LIN {X 0,Y 119.724,Z 602.099,A -85,B 0,C 180,E1 -25798.109,E2 -25798.109} C_VEL
LIN {X 0,Y 115.833,Z 604.315,A -85,B 0,C 180,E1 -25804.868,E2 -25804.868} C_VEL
LIN {X 0,Y 114.441,Z 604.822,A -85,B 0,C 180,E1 -25808.379,E2 -25808.379} C_VEL
LIN {X 0,Y 113.363,Z 604.891,A -85,B 0,C 180,E1 -25811.943,E2 -25811.943} C_VEL
LIN {X 0,Y 112.315,Z 603.854,A -85,B 0,C 180,E1 -25819.18,E2 -25819.18} C_VEL
LIN {X 0,Y 112.318,Z 602.743,A -85,B 0,C 180,E1 -25822.811,E2 -25822.811} C_VEL
LIN {X 0,Y 112.71,Z 601.178,A -85,B 0,C 180,E1 -25826.425,E2 -25826.425} C_VEL
LIN {X 0,Y 113.504,Z 598.082,A -85,B 0,C 180,E1 -25831.774,E2 -25831.774} C_VEL
LIN {X 0,Y 115.031,Z 593.941,A -85,B 0,C 180,E1 -25837.019,E2 -25837.019} C_VEL
LIN {X 0,Y 117.787,Z 587.628,A -85,B 0,C 180,E1 -25842.929,E2 -25842.929} C_VEL
LIN {X 0,Y 120.92,Z 580.766,A -85,B 0,C 180,E1 -25847.766,E2 -25847.766} C_VEL
LIN {X 0,Y 124.856,Z 572.161,A -85,B 0,C 180,E1 -25852.33,E2 -25852.33} C_VEL
LIN {X 0,Y 128.63,Z 563.345,A -85,B 0,C 180,E1 -25855.918,E2 -25855.918} C_VEL
LIN {X 0,Y 132.921,Z 552.472,A -85,B 0,C 180,E1 -25859.279,E2 -25859.279} C_VEL
LIN {X 0,Y 136.5,Z 541.503,A -85,B 0,C 180,E1 -25861.852,E2 -25861.852} C_VEL
LIN {X 0,Y 139.764,Z 529.243,A -85,B 0,C 180,E1 -25864.015,E2 -25864.015} C_VEL
LIN {X 0,Y 142.165,Z 517.629,A -85,B 0,C 180,E1 -25865.511,E2 -25865.511} C_VEL
LIN {X 0,Y 143.999,Z 504.981,A -85,B 0,C 180,E1 -25866.631,E2 -25866.631} C_VEL
LIN {X 0,Y 145.261,Z 489.73,A -85,B 0,C 180,E1 -25867.417,E2 -25867.417} C_VEL
LIN {X 0,Y 147.355,Z 457.951,A -85,B 0,C 180,E1 -25868.753,E2 -25868.753} C_VEL
LIN {X 0,Y 142.937,Z 448.506,A -85,B 0,C 180,E1 -25871.155,E2 -25871.155} C_VEL
LIN {X 0,Y 138.396,Z 440.269,A -85,B 0,C 180,E1 -25873.793,E2 -25873.793} C_VEL
LIN {X 0,Y 132.869,Z 431.292,A -85,B 0,C 180,E1 -25877.377,E2 -25877.377} C_VEL
LIN {X 0,Y 128.994,Z 425.855,A -85,B 0,C 180,E1 -25880.194,E2 -25880.194} C_VEL
LIN {X 0,Y 126.809,Z 422.709,A -85,B 0,C 180,E1 -25881.964,E2 -25881.964} C_VEL
LIN {X 0,Y 124.311,Z 419.474,A -85,B 0,C 180,E1 -25884.142,E2 -25884.142} C_VEL
LIN {X 0,Y 123.333,Z 418.034,A -85,B 0,C 180,E1 -25885.079,E2 -25885.079} C_VEL
LIN {X 0,Y 120.711,Z 415.377,A -85,B 0,C 180,E1 -25887.661,E2 -25887.661} C_VEL
LIN {X 0,Y 119.493,Z 412.941,A -85,B 0,C 180,E1 -25889.14,E2 -25889.14} C_VEL
LIN {X 0,Y 116.855,Z 411.214,A -85,B 0,C 180,E1 -25892.217,E2 -25892.217} C_VEL
LIN {X 0,Y 115.382,Z 409.029,A -85,B 0,C 180,E1 -25894.399,E2 -25894.399} C_VEL
LIN {X 0,Y 114.918,Z 407.137,A -85,B 0,C 180,E1 -25895.48,E2 -25895.48} C_VEL
LIN {X 0,Y 114.999,Z 407.157,A -85,B 0,C 180,E1 -25898.488,E2 -25898.488} C_VEL
LIN {X 0,Y 115.147,Z 407.106,A -85,B 0,C 180,E1 -25905.868,E2 -25905.868} C_VEL
LIN {X 0,Y 115.383,Z 407.111,A -85,B 0,C 180,E1 -25909.47,E2 -25909.47} C_VEL
LIN {X 0,Y 115.525,Z 407.056,A -85,B 0,C 180,E1 -25916.511,E2 -25916.511} C_VEL
LIN {X 0,Y 115.992,Z 407.035,A -85,B 0,C 180,E1 -25919.999,E2 -25919.999} C_VEL
LIN {X 0,Y 115.386,Z 407.107,A -85,B 0,C 180,E1 -25926.996,E2 -25926.996} C_VEL
LIN {X 0,Y 115.282,Z 407.118,A -85,B 0,C 180,E1 -25932.737,E2 -25932.737} C_VEL
LIN {X 0,Y 115.102,Z 407.186,A -85,B 0,C 180,E1 -25935.266,E2 -25935.266} C_VEL
LIN {X 0,Y 115.765,Z 409.428,A -85,B 0,C 180,E1 -25936.533,E2 -25936.533} C_VEL
LIN {X 0,Y 117.512,Z 411.742,A -85,B 0,C 180,E1 -25938.977,E2 -25938.977} C_VEL
LIN {X 0,Y 119.662,Z 413.079,A -85,B 0,C 180,E1 -25941.406,E2 -25941.406} C_VEL
LIN {X 0,Y 121.217,Z 416.052,A -85,B 0,C 180,E1 -25943.241,E2 -25943.241} C_VEL
LIN {X 0,Y 123.842,Z 418.627,A -85,B 0,C 180,E1 -25945.752,E2 -25945.752} C_VEL
LIN {X 0,Y 126.211,Z 422.141,A -85,B 0,C 180,E1 -25947.91,E2 -25947.91} C_VEL
LIN {X 0,Y 127.644,Z 423.794,A -85,B 0,C 180,E1 -25949.072,E2 -25949.072} C_VEL
LIN {X 0,Y 133.069,Z 431.531,A -85,B 0,C 180,E1 -25953.113,E2 -25953.113} C_VEL
LIN {X 0,Y 135.417,Z 435.627,A -85,B 0,C 180,E1 -25954.72,E2 -25954.72} C_VEL
LIN {X 0,Y 139.89,Z 445.297,A -85,B 0,C 180,E1 -25957.641,E2 -25957.641} C_VEL
LIN {X 0,Y 143.764,Z 455.4,A -85,B 0,C 180,E1 -25960.032,E2 -25960.032} C_VEL
LIN {X 0,Y 145.961,Z 461.997,A -85,B 0,C 180,E1 -25961.35,E2 -25961.35} C_VEL
LIN {X 0,Y 146.48,Z 475.088,A -85,B 0,C 180,E1 -25962.418,E2 -25962.418} C_VEL
LIN {X 0,Y 143.833,Z 511.707,A -85,B 0,C 180,E1 -25963.987,E2 -25963.987} C_VEL
LIN {X 0,Y 141.833,Z 525.299,A -85,B 0,C 180,E1 -25965.008,E2 -25965.008} C_VEL
LIN {X 0,Y 139.153,Z 538.159,A -85,B 0,C 180,E1 -25966.518,E2 -25966.518} C_VEL
LIN {X 0,Y 135.501,Z 550.822,A -85,B 0,C 180,E1 -25968.602,E2 -25968.602} C_VEL
LIN {X 0,Y 131.606,Z 562.106,A -85,B 0,C 180,E1 -25971.137,E2 -25971.137} C_VEL
LIN {X 0,Y 128.058,Z 571.239,A -85,B 0,C 180,E1 -25973.846,E2 -25973.846} C_VEL
LIN {X 0,Y 124.131,Z 580.605,A -85,B 0,C 180,E1 -25977.462,E2 -25977.462} C_VEL
LIN {X 0,Y 120.672,Z 588.035,A -85,B 0,C 180,E1 -25981.103,E2 -25981.103} C_VEL
LIN {X 0,Y 119.023,Z 592.301,A -85,B 0,C 180,E1 -25983.714,E2 -25983.714} C_VEL
LIN {X 0,Y 116.084,Z 599.069,A -85,B 0,C 180,E1 -25988.7,E2 -25988.7} C_VEL
LIN {X 0,Y 113.919,Z 604.457,A -85,B 0,C 180,E1 -25993.882,E2 -25993.882} C_VEL
LIN {X 0,Y 112.781,Z 608.657,A -85,B 0,C 180,E1 -25999.226,E2 -25999.226} C_VEL
LIN {X 0,Y 112.429,Z 610.864,A -85,B 0,C 180,E1 -26002.818,E2 -26002.818} C_VEL
LIN {X 0,Y 112.472,Z 613.501,A -85,B 0,C 180,E1 -26008.801,E2 -26008.801} C_VEL
LIN {X 0,Y 112.48,Z 614.275,A -85,B 0,C 180,E1 -26011.386,E2 -26011.386} C_VEL
LIN {X 0,Y 112.406,Z 615.185,A -85,B 0,C 180,E1 -26017.183,E2 -26017.183} C_VEL
LIN {X 0,Y 113.533,Z 614.858,A -85,B 0,C 180,E1 -26024.336,E2 -26024.336} C_VEL
LIN {X 0,Y 116.286,Z 613.013,A -85,B 0,C 180,E1 -26031.261,E2 -26031.261} C_VEL
LIN {X 0,Y 118.378,Z 611.46,A -85,B 0,C 180,E1 -26034.556,E2 -26034.556} C_VEL
LIN {X 0,Y 122.171,Z 608.364,A -85,B 0,C 180,E1 -26039.272,E2 -26039.272} C_VEL
LIN {X 0,Y 126.647,Z 604.233,A -85,B 0,C 180,E1 -26043.705,E2 -26043.705} C_VEL
LIN {X 0,Y 132.788,Z 597.948,A -85,B 0,C 180,E1 -26048.453,E2 -26048.453} C_VEL
LIN {X 0,Y 138.847,Z 591.139,A -85,B 0,C 180,E1 -26052.118,E2 -26052.118} C_VEL
LIN {X 0,Y 145.543,Z 582.699,A -85,B 0,C 180,E1 -26055.417,E2 -26055.417} C_VEL
LIN {X 0,Y 149.922,Z 576.362,A -85,B 0,C 180,E1 -26057.334,E2 -26057.334} C_VEL
LIN {X 0,Y 152.189,Z 572.121,A -85,B 0,C 180,E1 -26058.65,E2 -26058.65} C_VEL
LIN {X 0,Y 154.612,Z 564.94,A -85,B 0,C 180,E1 -26061.056,E2 -26061.056} C_VEL
LIN {X 0,Y 157,Z 557.347,A -85,B 0,C 180,E1 -26063.208,E2 -26063.208} C_VEL
LIN {X 0,Y 159.067,Z 552.385,A -85,B 0,C 180,E1 -26064.096,E2 -26064.096} C_VEL
LIN {X 0,Y 163.464,Z 541.938,A -85,B 0,C 180,E1 -26065.301,E2 -26065.301} C_VEL
LIN {X 0,Y 167.616,Z 528.948,A -85,B 0,C 180,E1 -26066.412,E2 -26066.412} C_VEL
LIN {X 0,Y 170.651,Z 515.665,A -85,B 0,C 180,E1 -26067.17,E2 -26067.17} C_VEL
LIN {X 0,Y 172.45,Z 501.424,A -85,B 0,C 180,E1 -26067.708,E2 -26067.708} C_VEL
LIN {X 0,Y 173.013,Z 494.554,A -85,B 0,C 180,E1 -26067.954,E2 -26067.954} C_VEL
LIN {X 0,Y 170.311,Z 486.612,A -85,B 0,C 180,E1 -26070.456,E2 -26070.456} C_VEL
LIN {X 0,Y 167.548,Z 479.336,A -85,B 0,C 180,E1 -26073.281,E2 -26073.281} C_VEL
LIN {X 0,Y 164.901,Z 473.089,A -85,B 0,C 180,E1 -26076.358,E2 -26076.358} C_VEL
LIN {X 0,Y 163.115,Z 469.142,A -85,B 0,C 180,E1 -26078.754,E2 -26078.754} C_VEL
LIN {X 0,Y 161.432,Z 465.461,A -85,B 0,C 180,E1 -26081.437,E2 -26081.437} C_VEL
LIN {X 0,Y 159.457,Z 461.943,A -85,B 0,C 180,E1 -26085.321,E2 -26085.321} C_VEL
LIN {X 0,Y 157.56,Z 458.915,A -85,B 0,C 180,E1 -26091.585,E2 -26091.585} C_VEL
LIN {X 0,Y 157.403,Z 457.318,A -85,B 0,C 180,E1 -26093.913,E2 -26093.913} C_VEL
LIN {X 0,Y 157.452,Z 457.311,A -85,B 0,C 180,E1 -26098.242,E2 -26098.242} C_VEL
LIN {X 0,Y 158.168,Z 460.156,A -85,B 0,C 180,E1 -26102.866,E2 -26102.866} C_VEL
LIN {X 0,Y 159.703,Z 462.142,A -85,B 0,C 180,E1 -26106.872,E2 -26106.872} C_VEL
LIN {X 0,Y 161.855,Z 465.875,A -85,B 0,C 180,E1 -26110.885,E2 -26110.885} C_VEL
LIN {X 0,Y 164.763,Z 470.847,A -85,B 0,C 180,E1 -26114.909,E2 -26114.909} C_VEL
LIN {X 0,Y 167.976,Z 476.505,A -85,B 0,C 180,E1 -26118.447,E2 -26118.447} C_VEL
LIN {X 0,Y 171.867,Z 484.181,A -85,B 0,C 180,E1 -26122.068,E2 -26122.068} C_VEL
LIN {X 0,Y 173.655,Z 487.825,A -85,B 0,C 180,E1 -26123.547,E2 -26123.547} C_VEL
LIN {X 0,Y 171.648,Z 505.752,A -85,B 0,C 180,E1 -26124.149,E2 -26124.149} C_VEL
LIN {X 0,Y 169.153,Z 518.376,A -85,B 0,C 180,E1 -26124.898,E2 -26124.898} C_VEL
LIN {X 0,Y 165.902,Z 530.053,A -85,B 0,C 180,E1 -26125.956,E2 -26125.956} C_VEL
LIN {X 0,Y 161.185,Z 542.276,A -85,B 0,C 180,E1 -26127.331,E2 -26127.331} C_VEL
LIN {X 0,Y 155.867,Z 553.494,A -85,B 0,C 180,E1 -26129.121,E2 -26129.121} C_VEL
LIN {X 0,Y 149.784,Z 564.254,A -85,B 0,C 180,E1 -26131.565,E2 -26131.565} C_VEL
LIN {X 0,Y 142.871,Z 574.243,A -85,B 0,C 180,E1 -26134.52,E2 -26134.52} C_VEL
LIN {X 0,Y 135.956,Z 582.655,A -85,B 0,C 180,E1 -26137.973,E2 -26137.973} C_VEL
LIN {X 0,Y 129.605,Z 589.39,A -85,B 0,C 180,E1 -26141.79,E2 -26141.79} C_VEL
LIN {X 0,Y 122.902,Z 595.508,A -85,B 0,C 180,E1 -26146.671,E2 -26146.671} C_VEL
LIN {X 0,Y 118.952,Z 598.636,A -85,B 0,C 180,E1 -26150.183,E2 -26150.183} C_VEL
LIN {X 0,Y 113.625,Z 602.314,A -85,B 0,C 180,E1 -26156.175,E2 -26156.175} C_VEL
LIN {X 0,Y 109.314,Z 604.585,A -85,B 0,C 180,E1 -26163.254,E2 -26163.254} C_VEL
LIN {X 0,Y 107.764,Z 605.126,A -85,B 0,C 180,E1 -26166.965,E2 -26166.965} C_VEL
LIN {X 0,Y 106.529,Z 605.244,A -85,B 0,C 180,E1 -26170.74,E2 -26170.74} C_VEL
LIN {X 0,Y 105.256,Z 604.261,A -85,B 0,C 180,E1 -26178.445,E2 -26178.445} C_VEL
LIN {X 0,Y 105.215,Z 603.187,A -85,B 0,C 180,E1 -26182.323,E2 -26182.323} C_VEL
LIN {X 0,Y 105.623,Z 601.53,A -85,B 0,C 180,E1 -26186.469,E2 -26186.469} C_VEL
LIN {X 0,Y 106.418,Z 598.626,A -85,B 0,C 180,E1 -26191.892,E2 -26191.892} C_VEL
LIN {X 0,Y 107.978,Z 594.55,A -85,B 0,C 180,E1 -26197.479,E2 -26197.479} C_VEL
LIN {X 0,Y 110.881,Z 588.304,A -85,B 0,C 180,E1 -26203.75,E2 -26203.75} C_VEL
LIN {X 0,Y 114.203,Z 581.517,A -85,B 0,C 180,E1 -26208.849,E2 -26208.849} C_VEL
LIN {X 0,Y 118.356,Z 573.044,A -85,B 0,C 180,E1 -26213.629,E2 -26213.629} C_VEL
LIN {X 0,Y 122.3,Z 564.341,A -85,B 0,C 180,E1 -26217.369,E2 -26217.369} C_VEL
LIN {X 0,Y 126.807,Z 553.608,A -85,B 0,C 180,E1 -26220.84,E2 -26220.84} C_VEL
LIN {X 0,Y 130.552,Z 542.908,A -85,B 0,C 180,E1 -26223.489,E2 -26223.489} C_VEL
LIN {X 0,Y 133.996,Z 530.917,A -85,B 0,C 180,E1 -26225.696,E2 -26225.696} C_VEL
LIN {X 0,Y 136.757,Z 518.43,A -85,B 0,C 180,E1 -26227.376,E2 -26227.376} C_VEL
LIN {X 0,Y 138.732,Z 505.641,A -85,B 0,C 180,E1 -26228.548,E2 -26228.548} C_VEL
LIN {X 0,Y 140.079,Z 490.411,A -85,B 0,C 180,E1 -26229.35,E2 -26229.35} C_VEL
LIN {X 0,Y 142.145,Z 460.167,A -85,B 0,C 180,E1 -26230.653,E2 -26230.653} C_VEL
LIN {X 0,Y 136.989,Z 449.433,A -85,B 0,C 180,E1 -26233.748,E2 -26233.748} C_VEL
LIN {X 0,Y 131.458,Z 439.752,A -85,B 0,C 180,E1 -26237.429,E2 -26237.429} C_VEL
LIN {X 0,Y 126.488,Z 432.151,A -85,B 0,C 180,E1 -26241.226,E2 -26241.226} C_VEL
LIN {X 0,Y 123.79,Z 428.3,A -85,B 0,C 180,E1 -26243.567,E2 -26243.567} C_VEL
LIN {X 0,Y 121.022,Z 424.337,A -85,B 0,C 180,E1 -26246.267,E2 -26246.267} C_VEL
LIN {X 0,Y 118.456,Z 421.495,A -85,B 0,C 180,E1 -26249.006,E2 -26249.006} C_VEL
LIN {X 0,Y 117.423,Z 419.563,A -85,B 0,C 180,E1 -26250.336,E2 -26250.336} C_VEL
LIN {X 0,Y 114.841,Z 417.45,A -85,B 0,C 180,E1 -26253.66,E2 -26253.66} C_VEL
LIN {X 0,Y 113.329,Z 414.785,A -85,B 0,C 180,E1 -26256.21,E2 -26256.21} C_VEL
LIN {X 0,Y 113.093,Z 414.058,A -85,B 0,C 180,E1 -26256.706,E2 -26256.706} C_VEL
LIN {X 0,Y 109.899,Z 412.045,A -85,B 0,C 180,E1 -26263.276,E2 -26263.276} C_VEL
LIN {X 0,Y 108.506,Z 408.955,A -85,B 0,C 180,E1 -26269.267,E2 -26269.267} C_VEL
LIN {X 0,Y 108.308,Z 407.973,A -85,B 0,C 180,E1 -26271.604,E2 -26271.604} C_VEL
LIN {X 0,Y 108.942,Z 407.913,A -85,B 0,C 180,E1 -26279.999,E2 -26279.999} C_VEL
LIN {X 0,Y 108.709,Z 407.989,A -85,B 0,C 180,E1 -26281.504,E2 -26281.504} C_VEL
LIN {X 0,Y 109.004,Z 409.947,A -85,B 0,C 180,E1 -26283.696,E2 -26283.696} C_VEL
LIN {X 0,Y 110.739,Z 412.499,A -85,B 0,C 180,E1 -26289.128,E2 -26289.128} C_VEL
LIN {X 0,Y 113.317,Z 414.146,A -85,B 0,C 180,E1 -26294.012,E2 -26294.012} C_VEL
LIN {X 0,Y 114.695,Z 417.115,A -85,B 0,C 180,E1 -26296.462,E2 -26296.462} C_VEL
LIN {X 0,Y 117.165,Z 419.334,A -85,B 0,C 180,E1 -26299.718,E2 -26299.718} C_VEL
LIN {X 0,Y 117.801,Z 420.224,A -85,B 0,C 180,E1 -26300.517,E2 -26300.517} C_VEL
LIN {X 0,Y 119.997,Z 423.462,A -85,B 0,C 180,E1 -26303.072,E2 -26303.072} C_VEL
LIN {X 0,Y 121.56,Z 425.08,A -85,B 0,C 180,E1 -26304.638,E2 -26304.638} C_VEL
LIN {X 0,Y 124.09,Z 428.671,A -85,B 0,C 180,E1 -26307.055,E2 -26307.055} C_VEL
LIN {X 0,Y 127.529,Z 433.561,A -85,B 0,C 180,E1 -26309.961,E2 -26309.961} C_VEL
LIN {X 0,Y 131.302,Z 439.503,A -85,B 0,C 180,E1 -26312.816,E2 -26312.816} C_VEL
LIN {X 0,Y 135.896,Z 449.916,A -85,B 0,C 180,E1 -26316.12,E2 -26316.12} C_VEL
LIN {X 0,Y 139.521,Z 459.83,A -85,B 0,C 180,E1 -26318.561,E2 -26318.561} C_VEL
LIN {X 0,Y 141.018,Z 464.805,A -85,B 0,C 180,E1 -26319.567,E2 -26319.567} C_VEL
LIN {X 0,Y 141.393,Z 474.77,A -85,B 0,C 180,E1 -26320.433,E2 -26320.433} C_VEL
LIN {X 0,Y 138.654,Z 511.118,A -85,B 0,C 180,E1 -26322.009,E2 -26322.009} C_VEL
LIN {X 0,Y 136.608,Z 524.623,A -85,B 0,C 180,E1 -26323.026,E2 -26323.026} C_VEL
LIN {X 0,Y 133.793,Z 537.662,A -85,B 0,C 180,E1 -26324.569,E2 -26324.569} C_VEL
LIN {X 0,Y 130.243,Z 549.566,A -85,B 0,C 180,E1 -26326.529,E2 -26326.529} C_VEL
LIN {X 0,Y 126.158,Z 561.023,A -85,B 0,C 180,E1 -26329.114,E2 -26329.114} C_VEL
LIN {X 0,Y 121.919,Z 571.344,A -85,B 0,C 180,E1 -26332.232,E2 -26332.232} C_VEL
LIN {X 0,Y 117.386,Z 581.442,A -85,B 0,C 180,E1 -26336.373,E2 -26336.373} C_VEL
LIN {X 0,Y 113.758,Z 588.946,A -85,B 0,C 180,E1 -26340.381,E2 -26340.381} C_VEL
LIN {X 0,Y 110.882,Z 595.203,A -85,B 0,C 180,E1 -26344.67,E2 -26344.67} C_VEL
LIN {X 0,Y 108.543,Z 600.404,A -85,B 0,C 180,E1 -26349.139,E2 -26349.139} C_VEL
LIN {X 0,Y 106.529,Z 605.431,A -85,B 0,C 180,E1 -26354.699,E2 -26354.699} C_VEL
LIN {X 0,Y 105.528,Z 609.313,A -85,B 0,C 180,E1 -26360.416,E2 -26360.416} C_VEL
LIN {X 0,Y 105.319,Z 612.142,A -85,B 0,C 180,E1 -26366.174,E2 -26366.174} C_VEL
LIN {X 0,Y 105.431,Z 613.706,A -85,B 0,C 180,E1 -26370.859,E2 -26370.859} C_VEL
LIN {X 0,Y 105.334,Z 614.829,A -85,B 0,C 180,E1 -26377.668,E2 -26377.668} C_VEL
LIN {X 0,Y 106.624,Z 614.557,A -85,B 0,C 180,E1 -26385.287,E2 -26385.287} C_VEL
LIN {X 0,Y 109.687,Z 612.766,A -85,B 0,C 180,E1 -26392.608,E2 -26392.608} C_VEL
LIN {X 0,Y 111.944,Z 611.255,A -85,B 0,C 180,E1 -26396.069,E2 -26396.069} C_VEL
LIN {X 0,Y 116.017,Z 608.209,A -85,B 0,C 180,E1 -26400.99,E2 -26400.99} C_VEL
LIN {X 0,Y 120.787,Z 604.132,A -85,B 0,C 180,E1 -26405.58,E2 -26405.58} C_VEL
LIN {X 0,Y 127.294,Z 597.911,A -85,B 0,C 180,E1 -26410.445,E2 -26410.445} C_VEL
LIN {X 0,Y 133.666,Z 591.171,A -85,B 0,C 180,E1 -26414.159,E2 -26414.159} C_VEL
LIN {X 0,Y 140.658,Z 582.836,A -85,B 0,C 180,E1 -26417.474,E2 -26417.474} C_VEL
LIN {X 0,Y 146.735,Z 574.286,A -85,B 0,C 180,E1 -26420.024,E2 -26420.024} C_VEL
LIN {X 0,Y 152.594,Z 564.928,A -85,B 0,C 180,E1 -26422.065,E2 -26422.065} C_VEL
LIN {X 0,Y 158.597,Z 553.347,A -85,B 0,C 180,E1 -26423.969,E2 -26423.969} C_VEL
LIN {X 0,Y 159.067,Z 552.385,A -85,B 0,C 180,E1 -26424.096,E2 -26424.096} C_VEL
LIN {X 0,Y 161.044,Z 547.315,A -85,B 0,C 180,E1 -26424.933,E2 -26424.933} C_VEL
LIN {X 0,Y 162.844,Z 538.909,A -85,B 0,C 180,E1 -26426.705,E2 -26426.705} C_VEL
LIN {X 0,Y 164.176,Z 530.173,A -85,B 0,C 180,E1 -26428.294,E2 -26428.294} C_VEL
LIN {X 0,Y 165.333,Z 524.59,A -85,B 0,C 180,E1 -26428.834,E2 -26428.834} C_VEL
LIN {X 0,Y 168.024,Z 511.325,A -85,B 0,C 180,E1 -26429.474,E2 -26429.474} C_VEL
LIN {X 0,Y 169.504,Z 497.365,A -85,B 0,C 180,E1 -26429.992,E2 -26429.992} C_VEL
LIN {X 0,Y 166.672,Z 488.688,A -85,B 0,C 180,E1 -26432.977,E2 -26432.977} C_VEL
LIN {X 0,Y 164.078,Z 481.812,A -85,B 0,C 180,E1 -26436.049,E2 -26436.049} C_VEL
LIN {X 0,Y 161.538,Z 475.581,A -85,B 0,C 180,E1 -26439.632,E2 -26439.632} C_VEL
LIN {X 0,Y 160.02,Z 472.053,A -85,B 0,C 180,E1 -26442.253,E2 -26442.253} C_VEL
LIN {X 0,Y 158.321,Z 468.793,A -85,B 0,C 180,E1 -26445.869,E2 -26445.869} C_VEL
LIN {X 0,Y 156.59,Z 465.711,A -85,B 0,C 180,E1 -26452.263,E2 -26452.263} C_VEL
LIN {X 0,Y 156.501,Z 464.314,A -85,B 0,C 180,E1 -26454.363,E2 -26454.363} C_VEL
LIN {X 0,Y 156.543,Z 464.375,A -85,B 0,C 180,E1 -26457.91,E2 -26457.91} C_VEL
LIN {X 0,Y 157.286,Z 467.301,A -85,B 0,C 180,E1 -26462.882,E2 -26462.882} C_VEL
LIN {X 0,Y 158.545,Z 469.038,A -85,B 0,C 180,E1 -26466.323,E2 -26466.323} C_VEL
LIN {X 0,Y 160.992,Z 473.561,A -85,B 0,C 180,E1 -26471.041,E2 -26471.041} C_VEL
LIN {X 0,Y 163.349,Z 477.854,A -85,B 0,C 180,E1 -26474.403,E2 -26474.403} C_VEL
LIN {X 0,Y 165.985,Z 482.743,A -85,B 0,C 180,E1 -26477.48,E2 -26477.48} C_VEL
LIN {X 0,Y 169.849,Z 490.775,A -85,B 0,C 180,E1 -26481.307,E2 -26481.307} C_VEL
LIN {X 0,Y 170.078,Z 491.288,A -85,B 0,C 180,E1 -26481.515,E2 -26481.515} C_VEL
LIN {X 0,Y 168.248,Z 506.682,A -85,B 0,C 180,E1 -26482.061,E2 -26482.061} C_VEL
LIN {X 0,Y 165.49,Z 519.773,A -85,B 0,C 180,E1 -26482.854,E2 -26482.854} C_VEL
LIN {X 0,Y 161.589,Z 532.682,A -85,B 0,C 180,E1 -26484.03,E2 -26484.03} C_VEL
LIN {X 0,Y 156.586,Z 544.701,A -85,B 0,C 180,E1 -26485.413,E2 -26485.413} C_VEL
LIN {X 0,Y 151.139,Z 555.426,A -85,B 0,C 180,E1 -26487.215,E2 -26487.215} C_VEL
LIN {X 0,Y 145.295,Z 565.193,A -85,B 0,C 180,E1 -26489.466,E2 -26489.466} C_VEL
LIN {X 0,Y 138.901,Z 574.037,A -85,B 0,C 180,E1 -26492.061,E2 -26492.061} C_VEL
LIN {X 0,Y 132.788,Z 581.297,A -85,B 0,C 180,E1 -26494.881,E2 -26494.881} C_VEL
LIN {X 0,Y 125.962,Z 588.375,A -85,B 0,C 180,E1 -26498.638,E2 -26498.638} C_VEL
LIN {X 0,Y 119.694,Z 593.986,A -85,B 0,C 180,E1 -26502.783,E2 -26502.783} C_VEL
LIN {X 0,Y 112.982,Z 599.115,A -85,B 0,C 180,E1 -26508.286,E2 -26508.286} C_VEL
LIN {X 0,Y 107.668,Z 602.52,A -85,B 0,C 180,E1 -26514.023,E2 -26514.023} C_VEL
LIN {X 0,Y 105.087,Z 603.896,A -85,B 0,C 180,E1 -26517.655,E2 -26517.655} C_VEL
LIN {X 0,Y 101.137,Z 605.425,A -85,B 0,C 180,E1 -26525.359,E2 -26525.359} C_VEL
LIN {X 0,Y 99.756,Z 605.593,A -85,B 0,C 180,E1 -26529.375,E2 -26529.375} C_VEL
LIN {X 0,Y 98.23,Z 604.666,A -85,B 0,C 180,E1 -26537.606,E2 -26537.606} C_VEL
LIN {X 0,Y 98.098,Z 603.621,A -85,B 0,C 180,E1 -26541.762,E2 -26541.762} C_VEL
LIN {X 0,Y 98.557,Z 601.8,A -85,B 0,C 180,E1 -26546.706,E2 -26546.706} C_VEL
LIN {X 0,Y 99.734,Z 597.928,A -85,B 0,C 180,E1 -26554.041,E2 -26554.041} C_VEL
LIN {X 0,Y 101.742,Z 593.539,A -85,B 0,C 180,E1 -26559.944,E2 -26559.944} C_VEL
LIN {X 0,Y 104.563,Z 587.968,A -85,B 0,C 180,E1 -26565.596,E2 -26565.596} C_VEL
LIN {X 0,Y 108.196,Z 581.018,A -85,B 0,C 180,E1 -26570.931,E2 -26570.931} C_VEL
LIN {X 0,Y 112.664,Z 572.304,A -85,B 0,C 180,E1 -26575.89,E2 -26575.89} C_VEL
LIN {X 0,Y 117.469,Z 562.399,A -85,B 0,C 180,E1 -26580.07,E2 -26580.07} C_VEL
LIN {X 0,Y 121.786,Z 552.312,A -85,B 0,C 180,E1 -26583.244,E2 -26583.244} C_VEL
LIN {X 0,Y 125.75,Z 541.145,A -85,B 0,C 180,E1 -26585.932,E2 -26585.932} C_VEL
LIN {X 0,Y 129.395,Z 528.612,A -85,B 0,C 180,E1 -26588.156,E2 -26588.156} C_VEL
LIN {X 0,Y 132.135,Z 515.841,A -85,B 0,C 180,E1 -26589.757,E2 -26589.757} C_VEL
LIN {X 0,Y 134.04,Z 502.589,A -85,B 0,C 180,E1 -26590.865,E2 -26590.865} C_VEL
LIN {X 0,Y 137.116,Z 462.643,A -85,B 0,C 180,E1 -26592.664,E2 -26592.664} C_VEL
LIN {X 0,Y 132.279,Z 452.521,A -85,B 0,C 180,E1 -26595.872,E2 -26595.872} C_VEL
LIN {X 0,Y 127.01,Z 443.147,A -85,B 0,C 180,E1 -26599.797,E2 -26599.797} C_VEL
LIN {X 0,Y 122.59,Z 436.291,A -85,B 0,C 180,E1 -26603.601,E2 -26603.601} C_VEL
LIN {X 0,Y 118.533,Z 430.395,A -85,B 0,C 180,E1 -26607.748,E2 -26607.748} C_VEL
LIN {X 0,Y 116.07,Z 427.256,A -85,B 0,C 180,E1 -26610.67,E2 -26610.67} C_VEL
LIN {X 0,Y 115.242,Z 425.978,A -85,B 0,C 180,E1 -26611.794,E2 -26611.794} C_VEL
LIN {X 0,Y 112.646,Z 423.291,A -85,B 0,C 180,E1 -26615.584,E2 -26615.584} C_VEL
LIN {X 0,Y 111.289,Z 420.722,A -85,B 0,C 180,E1 -26618.221,E2 -26618.221} C_VEL
LIN {X 0,Y 108.383,Z 418.413,A -85,B 0,C 180,E1 -26625.236,E2 -26625.236} C_VEL
LIN {X 0,Y 107.386,Z 415.152,A -85,B 0,C 180,E1 -26631.531,E2 -26631.531} C_VEL
LIN {X 0,Y 107.641,Z 415.015,A -85,B 0,C 180,E1 -26640.467,E2 -26640.467} C_VEL
LIN {X 0,Y 108.202,Z 417.518,A -85,B 0,C 180,E1 -26644.19,E2 -26644.19} C_VEL
LIN {X 0,Y 110.694,Z 420.251,A -85,B 0,C 180,E1 -26650.979,E2 -26650.979} C_VEL
LIN {X 0,Y 111.698,Z 420.937,A -85,B 0,C 180,E1 -26652.863,E2 -26652.863} C_VEL
LIN {X 0,Y 113.387,Z 424.156,A -85,B 0,C 180,E1 -26655.964,E2 -26655.964} C_VEL
LIN {X 0,Y 115.682,Z 426.457,A -85,B 0,C 180,E1 -26659.145,E2 -26659.145} C_VEL
LIN {X 0,Y 118.032,Z 429.953,A -85,B 0,C 180,E1 -26662.077,E2 -26662.077} C_VEL
LIN {X 0,Y 119.225,Z 431.369,A -85,B 0,C 180,E1 -26663.371,E2 -26663.371} C_VEL
LIN {X 0,Y 122.86,Z 436.682,A -85,B 0,C 180,E1 -26667.003,E2 -26667.003} C_VEL
LIN {X 0,Y 127.014,Z 443.083,A -85,B 0,C 180,E1 -26670.554,E2 -26670.554} C_VEL
LIN {X 0,Y 129.996,Z 449.489,A -85,B 0,C 180,E1 -26672.956,E2 -26672.956} C_VEL
LIN {X 0,Y 134.103,Z 460.315,A -85,B 0,C 180,E1 -26676.069,E2 -26676.069} C_VEL
LIN {X 0,Y 136.148,Z 466.88,A -85,B 0,C 180,E1 -26677.572,E2 -26677.572} C_VEL
LIN {X 0,Y 136.423,Z 475.585,A -85,B 0,C 180,E1 -26678.365,E2 -26678.365} C_VEL
LIN {X 0,Y 133.562,Z 511.236,A -85,B 0,C 180,E1 -26679.931,E2 -26679.931} C_VEL
LIN {X 0,Y 131.315,Z 525.207,A -85,B 0,C 180,E1 -26681.014,E2 -26681.014} C_VEL
LIN {X 0,Y 128.602,Z 537.144,A -85,B 0,C 180,E1 -26682.46,E2 -26682.46} C_VEL
LIN {X 0,Y 125.143,Z 548.291,A -85,B 0,C 180,E1 -26684.273,E2 -26684.273} C_VEL
LIN {X 0,Y 120.89,Z 559.933,A -85,B 0,C 180,E1 -26686.915,E2 -26686.915} C_VEL
LIN {X 0,Y 116.836,Z 569.316,A -85,B 0,C 180,E1 -26689.712,E2 -26689.712} C_VEL
LIN {X 0,Y 112.307,Z 578.955,A -85,B 0,C 180,E1 -26693.524,E2 -26693.524} C_VEL
LIN {X 0,Y 108.429,Z 586.489,A -85,B 0,C 180,E1 -26697.416,E2 -26697.416} C_VEL
LIN {X 0,Y 105.06,Z 593.396,A -85,B 0,C 180,E1 -26702.079,E2 -26702.079} C_VEL
LIN {X 0,Y 101.897,Z 599.804,A -85,B 0,C 180,E1 -26707.708,E2 -26707.708} C_VEL
LIN {X 0,Y 99.661,Z 604.888,A -85,B 0,C 180,E1 -26713.616,E2 -26713.616} C_VEL
LIN {X 0,Y 98.502,Z 608.823,A -85,B 0,C 180,E1 -26719.725,E2 -26719.725} C_VEL
LIN {X 0,Y 98.227,Z 611.702,A -85,B 0,C 180,E1 -26725.897,E2 -26725.897} C_VEL
LIN {X 0,Y 98.391,Z 613.048,A -85,B 0,C 180,E1 -26730,E2 -26730} C_VEL
LIN {X 0,Y 98.218,Z 613.953,A -85,B 0,C 180,E1 -26734.103,E2 -26734.103} C_VEL
LIN {X 0,Y 98.283,Z 614.464,A -85,B 0,C 180,E1 -26738.222,E2 -26738.222} C_VEL
LIN {X 0,Y 98.785,Z 614.562,A -85,B 0,C 180,E1 -26742.323,E2 -26742.323} C_VEL
LIN {X 0,Y 101.182,Z 613.573,A -85,B 0,C 180,E1 -26750.321,E2 -26750.321} C_VEL
LIN {X 0,Y 105.587,Z 611.051,A -85,B 0,C 180,E1 -26757.77,E2 -26757.77} C_VEL
LIN {X 0,Y 109.979,Z 608.049,A -85,B 0,C 180,E1 -26762.899,E2 -26762.899} C_VEL
LIN {X 0,Y 115.067,Z 604.022,A -85,B 0,C 180,E1 -26767.644,E2 -26767.644} C_VEL
LIN {X 0,Y 121.975,Z 597.877,A -85,B 0,C 180,E1 -26772.61,E2 -26772.61} C_VEL
LIN {X 0,Y 128.675,Z 591.204,A -85,B 0,C 180,E1 -26776.359,E2 -26776.359} C_VEL
LIN {X 0,Y 135.967,Z 582.948,A -85,B 0,C 180,E1 -26779.676,E2 -26779.676} C_VEL
LIN {X 0,Y 142.29,Z 574.519,A -85,B 0,C 180,E1 -26782.209,E2 -26782.209} C_VEL
LIN {X 0,Y 149.048,Z 564.12,A -85,B 0,C 180,E1 -26784.426,E2 -26784.426} C_VEL
LIN {X 0,Y 155.268,Z 552.437,A -85,B 0,C 180,E1 -26786.274,E2 -26786.274} C_VEL
LIN {X 0,Y 160.268,Z 540.796,A -85,B 0,C 180,E1 -26787.578,E2 -26787.578} C_VEL
LIN {X 0,Y 164.22,Z 528.73,A -85,B 0,C 180,E1 -26788.564,E2 -26788.564} C_VEL
LIN {X 0,Y 165.333,Z 524.59,A -85,B 0,C 180,E1 -26788.834,E2 -26788.834} C_VEL
LIN {X 0,Y 165.958,Z 520.826,A -85,B 0,C 180,E1 -26789.232,E2 -26789.232} C_VEL
LIN {X 0,Y 165.883,Z 514.975,A -85,B 0,C 180,E1 -26790.394,E2 -26790.394} C_VEL
LIN {X 0,Y 165.61,Z 509.069,A -85,B 0,C 180,E1 -26791.534,E2 -26791.534} C_VEL
LIN {X 0,Y 165.781,Z 505.212,A -85,B 0,C 180,E1 -26791.89,E2 -26791.89} C_VEL
LIN {X 0,Y 166.214,Z 500.224,A -85,B 0,C 180,E1 -26792.112,E2 -26792.112} C_VEL
LIN {X 0,Y 163.433,Z 491.491,A -85,B 0,C 180,E1 -26795.456,E2 -26795.456} C_VEL
LIN {X 0,Y 161.131,Z 485.147,A -85,B 0,C 180,E1 -26798.659,E2 -26798.659} C_VEL
LIN {X 0,Y 159.597,Z 481.125,A -85,B 0,C 180,E1 -26801.216,E2 -26801.216} C_VEL
LIN {X 0,Y 158.552,Z 478.497,A -85,B 0,C 180,E1 -26803.255,E2 -26803.255} C_VEL
LIN {X 0,Y 157.194,Z 475.69,A -85,B 0,C 180,E1 -26806.425,E2 -26806.425} C_VEL
LIN {X 0,Y 155.638,Z 472.465,A -85,B 0,C 180,E1 -26813.012,E2 -26813.012} C_VEL
LIN {X 0,Y 155.61,Z 471.301,A -85,B 0,C 180,E1 -26814.818,E2 -26814.818} C_VEL
LIN {X 0,Y 155.644,Z 471.406,A -85,B 0,C 180,E1 -26817.574,E2 -26817.574} C_VEL
LIN {X 0,Y 156.316,Z 474.284,A -85,B 0,C 180,E1 -26822.578,E2 -26822.578} C_VEL
LIN {X 0,Y 157.4,Z 475.945,A -85,B 0,C 180,E1 -26825.767,E2 -26825.767} C_VEL
LIN {X 0,Y 159.549,Z 480.165,A -85,B 0,C 180,E1 -26830.233,E2 -26830.233} C_VEL
LIN {X 0,Y 161.651,Z 484.22,A -85,B 0,C 180,E1 -26833.475,E2 -26833.475} C_VEL
LIN {X 0,Y 164.105,Z 489.11,A -85,B 0,C 180,E1 -26836.563,E2 -26836.563} C_VEL
LIN {X 0,Y 166.737,Z 494.932,A -85,B 0,C 180,E1 -26839.427,E2 -26839.427} C_VEL
LIN {X 0,Y 164.937,Z 508.395,A -85,B 0,C 180,E1 -26839.931,E2 -26839.931} C_VEL
LIN {X 0,Y 161.995,Z 521.369,A -85,B 0,C 180,E1 -26840.74,E2 -26840.74} C_VEL
LIN {X 0,Y 158.063,Z 533.695,A -85,B 0,C 180,E1 -26841.852,E2 -26841.852} C_VEL
LIN {X 0,Y 152.909,Z 545.521,A -85,B 0,C 180,E1 -26843.188,E2 -26843.188} C_VEL
LIN {X 0,Y 147.272,Z 556.159,A -85,B 0,C 180,E1 -26844.949,E2 -26844.949} C_VEL
LIN {X 0,Y 140.527,Z 566.846,A -85,B 0,C 180,E1 -26847.416,E2 -26847.416} C_VEL
LIN {X 0,Y 133.899,Z 575.428,A -85,B 0,C 180,E1 -26850.001,E2 -26850.001} C_VEL
LIN {X 0,Y 126.312,Z 583.741,A -85,B 0,C 180,E1 -26853.428,E2 -26853.428} C_VEL
LIN {X 0,Y 119.282,Z 590.4,A -85,B 0,C 180,E1 -26857.308,E2 -26857.308} C_VEL
LIN {X 0,Y 112.793,Z 595.67,A -85,B 0,C 180,E1 -26861.61,E2 -26861.61} C_VEL
LIN {X 0,Y 107.182,Z 599.577,A -85,B 0,C 180,E1 -26866.162,E2 -26866.162} C_VEL
LIN {X 0,Y 101.886,Z 602.712,A -85,B 0,C 180,E1 -26871.626,E2 -26871.626} C_VEL
LIN {X 0,Y 99.021,Z 604.142,A -85,B 0,C 180,E1 -26875.404,E2 -26875.404} C_VEL
LIN {X 0,Y 94.602,Z 605.725,A -85,B 0,C 180,E1 -26883.53,E2 -26883.53} C_VEL
LIN {X 0,Y 93.031,Z 605.93,A -85,B 0,C 180,E1 -26887.808,E2 -26887.808} C_VEL
LIN {X 0,Y 91.841,Z 605.706,A -85,B 0,C 180,E1 -26892.176,E2 -26892.176} C_VEL
LIN {X 0,Y 91.016,Z 604.051,A -85,B 0,C 180,E1 -26901.116,E2 -26901.116} C_VEL
LIN {X 0,Y 91.485,Z 602.025,A -85,B 0,C 180,E1 -26907.083,E2 -26907.083} C_VEL
LIN {X 0,Y 92.668,Z 598.466,A -85,B 0,C 180,E1 -26914.349,E2 -26914.349} C_VEL
LIN {X 0,Y 94.76,Z 594.14,A -85,B 0,C 180,E1 -26920.685,E2 -26920.685} C_VEL
LIN {X 0,Y 97.755,Z 588.635,A -85,B 0,C 180,E1 -26926.712,E2 -26926.712} C_VEL
LIN {X 0,Y 101.621,Z 581.774,A -85,B 0,C 180,E1 -26932.356,E2 -26932.356} C_VEL
LIN {X 0,Y 106.352,Z 573.175,A -85,B 0,C 180,E1 -26937.553,E2 -26937.553} C_VEL
LIN {X 0,Y 110.902,Z 564.353,A -85,B 0,C 180,E1 -26941.52,E2 -26941.52} C_VEL
LIN {X 0,Y 115.945,Z 553.481,A -85,B 0,C 180,E1 -26945.158,E2 -26945.158} C_VEL
LIN {X 0,Y 120.102,Z 542.523,A -85,B 0,C 180,E1 -26947.909,E2 -26947.909} C_VEL
LIN {X 0,Y 123.946,Z 530.254,A -85,B 0,C 180,E1 -26950.163,E2 -26950.163} C_VEL
LIN {X 0,Y 126.937,Z 517.474,A -85,B 0,C 180,E1 -26951.862,E2 -26951.862} C_VEL
LIN {X 0,Y 129.083,Z 503.863,A -85,B 0,C 180,E1 -26953.039,E2 -26953.039} C_VEL
LIN {X 0,Y 131.129,Z 480.069,A -85,B 0,C 180,E1 -26954.165,E2 -26954.165} C_VEL
LIN {X 0,Y 132.249,Z 465.212,A -85,B 0,C 180,E1 -26954.823,E2 -26954.823} C_VEL
LIN {X 0,Y 128.087,Z 456.27,A -85,B 0,C 180,E1 -26957.899,E2 -26957.899} C_VEL
LIN {X 0,Y 123.148,Z 447.353,A -85,B 0,C 180,E1 -26961.991,E2 -26961.991} C_VEL
LIN {X 0,Y 119.032,Z 440.626,A -85,B 0,C 180,E1 -26966.004,E2 -26966.004} C_VEL
LIN {X 0,Y 116.297,Z 436.622,A -85,B 0,C 180,E1 -26969.09,E2 -26969.09} C_VEL
LIN {X 0,Y 113.784,Z 433.016,A -85,B 0,C 180,E1 -26972.402,E2 -26972.402} C_VEL
LIN {X 0,Y 110.591,Z 429.068,A -85,B 0,C 180,E1 -26977.585,E2 -26977.585} C_VEL
LIN {X 0,Y 109.988,Z 427.655,A -85,B 0,C 180,E1 -26978.934,E2 -26978.934} C_VEL
LIN {X 0,Y 107.178,Z 425.065,A -85,B 0,C 180,E1 -26986.452,E2 -26986.452} C_VEL
LIN {X 0,Y 106.44,Z 422.071,A -85,B 0,C 180,E1 -26992.411,E2 -26992.411} C_VEL
LIN {X 0,Y 106.649,Z 422.116,A -85,B 0,C 180,E1 -26999.763,E2 -26999.763} C_VEL
LIN {X 0,Y 107.276,Z 424.736,A -85,B 0,C 180,E1 -27004.108,E2 -27004.108} C_VEL
LIN {X 0,Y 110.208,Z 427.79,A -85,B 0,C 180,E1 -27011.844,E2 -27011.844} C_VEL
LIN {X 0,Y 112.091,Z 431.179,A -85,B 0,C 180,E1 -27015.454,E2 -27015.454} C_VEL
LIN {X 0,Y 113.802,Z 433.031,A -85,B 0,C 180,E1 -27017.985,E2 -27017.985} C_VEL
LIN {X 0,Y 116.283,Z 436.663,A -85,B 0,C 180,E1 -27021.261,E2 -27021.261} C_VEL
LIN {X 0,Y 120.113,Z 442.355,A -85,B 0,C 180,E1 -27025.476,E2 -27025.476} C_VEL
LIN {X 0,Y 124.413,Z 449.453,A -85,B 0,C 180,E1 -27029.467,E2 -27029.467} C_VEL
LIN {X 0,Y 128.044,Z 458.608,A -85,B 0,C 180,E1 -27032.645,E2 -27032.645} C_VEL
LIN {X 0,Y 131.056,Z 467.89,A -85,B 0,C 180,E1 -27035.135,E2 -27035.135} C_VEL
LIN {X 0,Y 131.508,Z 469.525,A -85,B 0,C 180,E1 -27035.508,E2 -27035.508} C_VEL
LIN {X 0,Y 131.575,Z 476.903,A -85,B 0,C 180,E1 -27036.154,E2 -27036.154} C_VEL
LIN {X 0,Y 128.746,Z 510.785,A -85,B 0,C 180,E1 -27037.664,E2 -27037.664} C_VEL
LIN {X 0,Y 126.417,Z 524.67,A -85,B 0,C 180,E1 -27038.731,E2 -27038.731} C_VEL
LIN {X 0,Y 123.3,Z 537.633,A -85,B 0,C 180,E1 -27040.328,E2 -27040.328} C_VEL
LIN {X 0,Y 119.14,Z 550.203,A -85,B 0,C 180,E1 -27042.494,E2 -27042.494} C_VEL
LIN {X 0,Y 114.648,Z 561.416,A -85,B 0,C 180,E1 -27045.175,E2 -27045.175} C_VEL
LIN {X 0,Y 110.507,Z 570.497,A -85,B 0,C 180,E1 -27048.105,E2 -27048.105} C_VEL
LIN {X 0,Y 105.759,Z 579.8,A -85,B 0,C 180,E1 -27052.072,E2 -27052.072} C_VEL
LIN {X 0,Y 100.752,Z 588.835,A -85,B 0,C 180,E1 -27057.276,E2 -27057.276} C_VEL
LIN {X 0,Y 98.125,Z 593.867,A -85,B 0,C 180,E1 -27061.09,E2 -27061.09} C_VEL
LIN {X 0,Y 95.328,Z 599.196,A -85,B 0,C 180,E1 -27066.079,E2 -27066.079} C_VEL
LIN {X 0,Y 92.838,Z 604.341,A -85,B 0,C 180,E1 -27072.374,E2 -27072.374} C_VEL
LIN {X 0,Y 91.502,Z 608.33,A -85,B 0,C 180,E1 -27078.93,E2 -27078.93} C_VEL
LIN {X 0,Y 91.119,Z 611.258,A -85,B 0,C 180,E1 -27085.576,E2 -27085.576} C_VEL
LIN {X 0,Y 91.303,Z 612.631,A -85,B 0,C 180,E1 -27090,E2 -27090} C_VEL
LIN {X 0,Y 91.118,Z 613.559,A -85,B 0,C 180,E1 -27094.424,E2 -27094.424} C_VEL
LIN {X 0,Y 91.258,Z 614.094,A -85,B 0,C 180,E1 -27098.86,E2 -27098.86} C_VEL
LIN {X 0,Y 91.833,Z 614.235,A -85,B 0,C 180,E1 -27103.273,E2 -27103.273} C_VEL
LIN {X 0,Y 94.523,Z 613.297,A -85,B 0,C 180,E1 -27111.824,E2 -27111.824} C_VEL
LIN {X 0,Y 99.324,Z 610.838,A -85,B 0,C 180,E1 -27119.689,E2 -27119.689} C_VEL
LIN {X 0,Y 104.056,Z 607.876,A -85,B 0,C 180,E1 -27125.035,E2 -27125.035} C_VEL
LIN {X 0,Y 109.518,Z 603.901,A -85,B 0,C 180,E1 -27129.919,E2 -27129.919} C_VEL
LIN {X 0,Y 115.721,Z 598.819,A -85,B 0,C 180,E1 -27134.299,E2 -27134.299} C_VEL
LIN {X 0,Y 122.677,Z 592.467,A -85,B 0,C 180,E1 -27138.136,E2 -27138.136} C_VEL
LIN {X 0,Y 130.19,Z 584.545,A -85,B 0,C 180,E1 -27141.511,E2 -27141.511} C_VEL
LIN {X 0,Y 136.733,Z 576.501,A -85,B 0,C 180,E1 -27144.049,E2 -27144.049} C_VEL
LIN {X 0,Y 143.605,Z 566.708,A -85,B 0,C 180,E1 -27146.3,E2 -27146.3} C_VEL
LIN {X 0,Y 150.017,Z 555.796,A -85,B 0,C 180,E1 -27148.114,E2 -27148.114} C_VEL
LIN {X 0,Y 155.863,Z 543.356,A -85,B 0,C 180,E1 -27149.581,E2 -27149.581} C_VEL
LIN {X 0,Y 160.286,Z 531.161,A -85,B 0,C 180,E1 -27150.625,E2 -27150.625} C_VEL
LIN {X 0,Y 163.518,Z 519.067,A -85,B 0,C 180,E1 -27151.322,E2 -27151.322} C_VEL
LIN {X 0,Y 165.781,Z 505.212,A -85,B 0,C 180,E1 -27151.89,E2 -27151.89} C_VEL
LIN {X 0,Y 165.712,Z 502.716,A -85,B 0,C 180,E1 -27152.247,E2 -27152.247} C_VEL
LIN {X 0,Y 164.977,Z 500.411,A -85,B 0,C 180,E1 -27153.109,E2 -27153.109} C_VEL
LIN {X 0,Y 163.81,Z 498.736,A -85,B 0,C 180,E1 -27154.289,E2 -27154.289} C_VEL
LIN {X 0,Y 160.931,Z 495.58,A -85,B 0,C 180,E1 -27157.404,E2 -27157.404} C_VEL
LIN {X 0,Y 160.459,Z 494.428,A -85,B 0,C 180,E1 -27158.069,E2 -27158.069} C_VEL
LIN {X 0,Y 158.378,Z 488.241,A -85,B 0,C 180,E1 -27161.653,E2 -27161.653} C_VEL
LIN {X 0,Y 157.284,Z 485.225,A -85,B 0,C 180,E1 -27163.95,E2 -27163.95} C_VEL
LIN {X 0,Y 155.967,Z 482.431,A -85,B 0,C 180,E1 -27167.311,E2 -27167.311} C_VEL
LIN {X 0,Y 154.717,Z 479.185,A -85,B 0,C 180,E1 -27173.785,E2 -27173.785} C_VEL
LIN {X 0,Y 154.726,Z 478.481,A -85,B 0,C 180,E1 -27174.788,E2 -27174.788} C_VEL
LIN {X 0,Y 154.745,Z 478.733,A -85,B 0,C 180,E1 -27177.631,E2 -27177.631} C_VEL
LIN {X 0,Y 155.77,Z 481.918,A -85,B 0,C 180,E1 -27183.719,E2 -27183.719} C_VEL
LIN {X 0,Y 156.262,Z 482.777,A -85,B 0,C 180,E1 -27185.161,E2 -27185.161} C_VEL
LIN {X 0,Y 158.192,Z 486.875,A -85,B 0,C 180,E1 -27189.51,E2 -27189.51} C_VEL
LIN {X 0,Y 160.265,Z 491.069,A -85,B 0,C 180,E1 -27192.908,E2 -27192.908} C_VEL
LIN {X 0,Y 162.884,Z 496.837,A -85,B 0,C 180,E1 -27196.378,E2 -27196.378} C_VEL
LIN {X 0,Y 163.611,Z 498.651,A -85,B 0,C 180,E1 -27197.283,E2 -27197.283} C_VEL
LIN {X 0,Y 161.441,Z 512.047,A -85,B 0,C 180,E1 -27197.824,E2 -27197.824} C_VEL
LIN {X 0,Y 158.292,Z 524.524,A -85,B 0,C 180,E1 -27198.659,E2 -27198.659} C_VEL
LIN {X 0,Y 154.016,Z 536.522,A -85,B 0,C 180,E1 -27199.758,E2 -27199.758} C_VEL
LIN {X 0,Y 148.724,Z 547.784,A -85,B 0,C 180,E1 -27201.049,E2 -27201.049} C_VEL
LIN {X 0,Y 143.062,Z 557.873,A -85,B 0,C 180,E1 -27202.755,E2 -27202.755} C_VEL
LIN {X 0,Y 137.336,Z 566.524,A -85,B 0,C 180,E1 -27204.727,E2 -27204.727} C_VEL
LIN {X 0,Y 130.427,Z 575.252,A -85,B 0,C 180,E1 -27207.243,E2 -27207.243} C_VEL
LIN {X 0,Y 122.468,Z 583.664,A -85,B 0,C 180,E1 -27210.596,E2 -27210.596} C_VEL
LIN {X 0,Y 115.032,Z 590.399,A -85,B 0,C 180,E1 -27214.434,E2 -27214.434} C_VEL
LIN {X 0,Y 108.109,Z 595.737,A -85,B 0,C 180,E1 -27218.732,E2 -27218.732} C_VEL
LIN {X 0,Y 101.54,Z 600.042,A -85,B 0,C 180,E1 -27223.801,E2 -27223.801} C_VEL
LIN {X 0,Y 96.311,Z 602.901,A -85,B 0,C 180,E1 -27228.949,E2 -27228.949} C_VEL
LIN {X 0,Y 93.143,Z 604.385,A -85,B 0,C 180,E1 -27232.87,E2 -27232.87} C_VEL
LIN {X 0,Y 88.175,Z 606.025,A -85,B 0,C 180,E1 -27241.431,E2 -27241.431} C_VEL
LIN {X 0,Y 86.371,Z 606.258,A -85,B 0,C 180,E1 -27245.994,E2 -27245.994} C_VEL
LIN {X 0,Y 85.012,Z 606.085,A -85,B 0,C 180,E1 -27250.69,E2 -27250.69} C_VEL
LIN {X 0,Y 83.933,Z 604.483,A -85,B 0,C 180,E1 -27260.36,E2 -27260.36} C_VEL
LIN {X 0,Y 84.427,Z 602.304,A -85,B 0,C 180,E1 -27267.378,E2 -27267.378} C_VEL
LIN {X 0,Y 85.604,Z 599.005,A -85,B 0,C 180,E1 -27274.709,E2 -27274.709} C_VEL
LIN {X 0,Y 87.78,Z 594.742,A -85,B 0,C 180,E1 -27281.546,E2 -27281.546} C_VEL
LIN {X 0,Y 91.627,Z 588.295,A -85,B 0,C 180,E1 -27289.025,E2 -27289.025} C_VEL
LIN {X 0,Y 95.898,Z 581.231,A -85,B 0,C 180,E1 -27294.922,E2 -27294.922} C_VEL
LIN {X 0,Y 101.052,Z 572.423,A -85,B 0,C 180,E1 -27300.279,E2 -27300.279} C_VEL
LIN {X 0,Y 105.98,Z 563.382,A -85,B 0,C 180,E1 -27304.309,E2 -27304.309} C_VEL
LIN {X 0,Y 110.797,Z 553.396,A -85,B 0,C 180,E1 -27307.626,E2 -27307.626} C_VEL
LIN {X 0,Y 115.187,Z 542.327,A -85,B 0,C 180,E1 -27310.41,E2 -27310.41} C_VEL
LIN {X 0,Y 119.238,Z 529.922,A -85,B 0,C 180,E1 -27312.672,E2 -27312.672} C_VEL
LIN {X 0,Y 122.235,Z 517.579,A -85,B 0,C 180,E1 -27314.292,E2 -27314.292} C_VEL
LIN {X 0,Y 124.422,Z 504.294,A -85,B 0,C 180,E1 -27315.448,E2 -27315.448} C_VEL
LIN {X 0,Y 126.526,Z 481.21,A -85,B 0,C 180,E1 -27316.543,E2 -27316.543} C_VEL
LIN {X 0,Y 127.551,Z 467.731,A -85,B 0,C 180,E1 -27317.169,E2 -27317.169} C_VEL
LIN {X 0,Y 123.817,Z 459.694,A -85,B 0,C 180,E1 -27320.258,E2 -27320.258} C_VEL
LIN {X 0,Y 120.024,Z 452.558,A -85,B 0,C 180,E1 -27323.772,E2 -27323.772} C_VEL
LIN {X 0,Y 116.401,Z 446.348,A -85,B 0,C 180,E1 -27327.671,E2 -27327.671} C_VEL
LIN {X 0,Y 113.967,Z 442.649,A -85,B 0,C 180,E1 -27330.692,E2 -27330.692} C_VEL
LIN {X 0,Y 111.497,Z 438.939,A -85,B 0,C 180,E1 -27334.318,E2 -27334.318} C_VEL
LIN {X 0,Y 108.989,Z 435.496,A -85,B 0,C 180,E1 -27338.917,E2 -27338.917} C_VEL
LIN {X 0,Y 108.495,Z 434.395,A -85,B 0,C 180,E1 -27340.117,E2 -27340.117} C_VEL
LIN {X 0,Y 106.012,Z 431.691,A -85,B 0,C 180,E1 -27347.749,E2 -27347.749} C_VEL
LIN {X 0,Y 105.561,Z 429.242,A -85,B 0,C 180,E1 -27352.347,E2 -27352.347} C_VEL
LIN {X 0,Y 105.685,Z 429.168,A -85,B 0,C 180,E1 -27359.088,E2 -27359.088} C_VEL
LIN {X 0,Y 106.381,Z 431.979,A -85,B 0,C 180,E1 -27364.143,E2 -27364.143} C_VEL
LIN {X 0,Y 108.728,Z 434.468,A -85,B 0,C 180,E1 -27370.709,E2 -27370.709} C_VEL
LIN {X 0,Y 110.582,Z 437.892,A -85,B 0,C 180,E1 -27374.546,E2 -27374.546} C_VEL
LIN {X 0,Y 111.929,Z 439.446,A -85,B 0,C 180,E1 -27376.705,E2 -27376.705} C_VEL
LIN {X 0,Y 115.185,Z 444.519,A -85,B 0,C 180,E1 -27381.239,E2 -27381.239} C_VEL
LIN {X 0,Y 117.948,Z 448.892,A -85,B 0,C 180,E1 -27384.425,E2 -27384.425} C_VEL
LIN {X 0,Y 121.325,Z 454.9,A -85,B 0,C 180,E1 -27387.841,E2 -27387.841} C_VEL
LIN {X 0,Y 124.75,Z 464.385,A -85,B 0,C 180,E1 -27391.17,E2 -27391.17} C_VEL
LIN {X 0,Y 127,Z 471.887,A -85,B 0,C 180,E1 -27393.243,E2 -27393.243} C_VEL
LIN {X 0,Y 127.025,Z 477.3,A -85,B 0,C 180,E1 -27393.746,E2 -27393.746} C_VEL
LIN {X 0,Y 124.134,Z 510.34,A -85,B 0,C 180,E1 -27395.219,E2 -27395.219} C_VEL
LIN {X 0,Y 121.759,Z 524.068,A -85,B 0,C 180,E1 -27396.267,E2 -27396.267} C_VEL
LIN {X 0,Y 118.488,Z 537.103,A -85,B 0,C 180,E1 -27397.852,E2 -27397.852} C_VEL
LIN {X 0,Y 114.401,Z 548.905,A -85,B 0,C 180,E1 -27399.835,E2 -27399.835} C_VEL
LIN {X 0,Y 109.737,Z 560.317,A -85,B 0,C 180,E1 -27402.567,E2 -27402.567} C_VEL
LIN {X 0,Y 105.261,Z 569.519,A -85,B 0,C 180,E1 -27405.489,E2 -27405.489} C_VEL
LIN {X 0,Y 100.202,Z 578.973,A -85,B 0,C 180,E1 -27409.552,E2 -27409.552} C_VEL
LIN {X 0,Y 95.622,Z 586.717,A -85,B 0,C 180,E1 -27413.987,E2 -27413.987} C_VEL
LIN {X 0,Y 91.946,Z 593.197,A -85,B 0,C 180,E1 -27418.94,E2 -27418.94} C_VEL
LIN {X 0,Y 88.858,Z 598.573,A -85,B 0,C 180,E1 -27424.215,E2 -27424.215} C_VEL
LIN {X 0,Y 86.053,Z 603.787,A -85,B 0,C 180,E1 -27430.933,E2 -27430.933} C_VEL
LIN {X 0,Y 84.506,Z 607.831,A -85,B 0,C 180,E1 -27438,E2 -27438} C_VEL
LIN {X 0,Y 84.043,Z 610.805,A -85,B 0,C 180,E1 -27445.203,E2 -27445.203} C_VEL
LIN {X 0,Y 84.195,Z 612.213,A -85,B 0,C 180,E1 -27450,E2 -27450} C_VEL
LIN {X 0,Y 84.041,Z 613.165,A -85,B 0,C 180,E1 -27454.797,E2 -27454.797} C_VEL
LIN {X 0,Y 84.921,Z 613.898,A -85,B 0,C 180,E1 -27464.375,E2 -27464.375} C_VEL
LIN {X 0,Y 87.938,Z 613.022,A -85,B 0,C 180,E1 -27473.553,E2 -27473.553} C_VEL
LIN {X 0,Y 93.19,Z 610.614,A -85,B 0,C 180,E1 -27481.863,E2 -27481.863} C_VEL
LIN {X 0,Y 98.298,Z 607.7,A -85,B 0,C 180,E1 -27487.424,E2 -27487.424} C_VEL
LIN {X 0,Y 104.159,Z 603.779,A -85,B 0,C 180,E1 -27492.433,E2 -27492.433} C_VEL
LIN {X 0,Y 110.751,Z 598.755,A -85,B 0,C 180,E1 -27496.865,E2 -27496.865} C_VEL
LIN {X 0,Y 118.058,Z 592.477,A -85,B 0,C 180,E1 -27500.703,E2 -27500.703} C_VEL
LIN {X 0,Y 125.891,Z 584.654,A -85,B 0,C 180,E1 -27504.043,E2 -27504.043} C_VEL
LIN {X 0,Y 134.086,Z 574.918,A -85,B 0,C 180,E1 -27506.993,E2 -27506.993} C_VEL
LIN {X 0,Y 141.294,Z 564.848,A -85,B 0,C 180,E1 -27509.093,E2 -27509.093} C_VEL
LIN {X 0,Y 147.89,Z 553.467,A -85,B 0,C 180,E1 -27510.832,E2 -27510.832} C_VEL
LIN {X 0,Y 153.169,Z 542.311,A -85,B 0,C 180,E1 -27512.036,E2 -27512.036} C_VEL
LIN {X 0,Y 157.712,Z 529.856,A -85,B 0,C 180,E1 -27513.028,E2 -27513.028} C_VEL
LIN {X 0,Y 160.974,Z 517.392,A -85,B 0,C 180,E1 -27513.701,E2 -27513.701} C_VEL
LIN {X 0,Y 163.095,Z 504.344,A -85,B 0,C 180,E1 -27514.196,E2 -27514.196} C_VEL
LIN {X 0,Y 163.13,Z 503.302,A -85,B 0,C 180,E1 -27514.31,E2 -27514.31} C_VEL
LIN {X 0,Y 161.079,Z 496.338,A -85,B 0,C 180,E1 -27517.143,E2 -27517.143} C_VEL
LIN {X 0,Y 160.459,Z 494.428,A -85,B 0,C 180,E1 -27518.069,E2 -27518.069} C_VEL
LIN {X 0,Y 159.668,Z 492.509,A -85,B 0,C 180,E1 -27519.261,E2 -27519.261} C_VEL
LIN {X 0,Y 158.344,Z 490.785,A -85,B 0,C 180,E1 -27521.246,E2 -27521.246} C_VEL
LIN {X 0,Y 156.225,Z 489.797,A -85,B 0,C 180,E1 -27524.818,E2 -27524.818} C_VEL
LIN {X 0,Y 154.914,Z 489.312,A -85,B 0,C 180,E1 -27527.8,E2 -27527.8} C_VEL
LIN {X 0,Y 154.465,Z 488.723,A -85,B 0,C 180,E1 -27529.293,E2 -27529.293} C_VEL
LIN {X 0,Y 153.825,Z 485.802,A -85,B 0,C 180,E1 -27534.758,E2 -27534.758} C_VEL
LIN {X 0,Y 153.851,Z 485.962,A -85,B 0,C 180,E1 -27537.618,E2 -27537.618} C_VEL
LIN {X 0,Y 155.112,Z 489.527,A -85,B 0,C 180,E1 -27544.452,E2 -27544.452} C_VEL
LIN {X 0,Y 156.846,Z 493.519,A -85,B 0,C 180,E1 -27548.739,E2 -27548.739} C_VEL
LIN {X 0,Y 158.615,Z 497.416,A -85,B 0,C 180,E1 -27551.907,E2 -27551.907} C_VEL
LIN {X 0,Y 160.63,Z 502.426,A -85,B 0,C 180,E1 -27555.023,E2 -27555.023} C_VEL
LIN {X 0,Y 158.096,Z 515.756,A -85,B 0,C 180,E1 -27555.654,E2 -27555.654} C_VEL
LIN {X 0,Y 154.642,Z 527.813,A -85,B 0,C 180,E1 -27556.509,E2 -27556.509} C_VEL
LIN {X 0,Y 150.188,Z 539.251,A -85,B 0,C 180,E1 -27557.557,E2 -27557.557} C_VEL
LIN {X 0,Y 144.784,Z 550.044,A -85,B 0,C 180,E1 -27558.821,E2 -27558.821} C_VEL
LIN {X 0,Y 138.997,Z 559.671,A -85,B 0,C 180,E1 -27560.453,E2 -27560.453} C_VEL
LIN {X 0,Y 131.585,Z 569.95,A -85,B 0,C 180,E1 -27562.882,E2 -27562.882} C_VEL
LIN {X 0,Y 124.456,Z 578.1,A -85,B 0,C 180,E1 -27565.379,E2 -27565.379} C_VEL
LIN {X 0,Y 116.631,Z 585.742,A -85,B 0,C 180,E1 -27568.636,E2 -27568.636} C_VEL
LIN {X 0,Y 108.564,Z 592.354,A -85,B 0,C 180,E1 -27572.696,E2 -27572.696} C_VEL
LIN {X 0,Y 101.405,Z 597.329,A -85,B 0,C 180,E1 -27577.155,E2 -27577.155} C_VEL
LIN {X 0,Y 94.876,Z 601.143,A -85,B 0,C 180,E1 -27582.206,E2 -27582.206} C_VEL
LIN {X 0,Y 90.967,Z 603.09,A -85,B 0,C 180,E1 -27585.948,E2 -27585.948} C_VEL
LIN {X 0,Y 87.469,Z 604.613,A -85,B 0,C 180,E1 -27590.001,E2 -27590.001} C_VEL
LIN {X 0,Y 84.433,Z 605.676,A -85,B 0,C 180,E1 -27594.363,E2 -27594.363} C_VEL
LIN {X 0,Y 81.741,Z 606.352,A -85,B 0,C 180,E1 -27599.296,E2 -27599.296} C_VEL
LIN {X 0,Y 78.252,Z 606.454,A -85,B 0,C 180,E1 -27608.946,E2 -27608.946} C_VEL
LIN {X 0,Y 77.272,Z 605.883,A -85,B 0,C 180,E1 -27614.166,E2 -27614.166} C_VEL
LIN {X 0,Y 76.858,Z 604.915,A -85,B 0,C 180,E1 -27619.463,E2 -27619.463} C_VEL
LIN {X 0,Y 77.369,Z 602.571,A -85,B 0,C 180,E1 -27627.765,E2 -27627.765} C_VEL
LIN {X 0,Y 78.542,Z 599.544,A -85,B 0,C 180,E1 -27635.134,E2 -27635.134} C_VEL
LIN {X 0,Y 80.825,Z 595.345,A -85,B 0,C 180,E1 -27642.555,E2 -27642.555} C_VEL
LIN {X 0,Y 84.956,Z 588.963,A -85,B 0,C 180,E1 -27650.584,E2 -27650.584} C_VEL
LIN {X 0,Y 89.534,Z 582.009,A -85,B 0,C 180,E1 -27656.83,E2 -27656.83} C_VEL
LIN {X 0,Y 95.003,Z 573.295,A -85,B 0,C 180,E1 -27662.433,E2 -27662.433} C_VEL
LIN {X 0,Y 100.769,Z 563.386,A -85,B 0,C 180,E1 -27666.979,E2 -27666.979} C_VEL
LIN {X 0,Y 105.864,Z 553.298,A -85,B 0,C 180,E1 -27670.335,E2 -27670.335} C_VEL
LIN {X 0,Y 110.499,Z 542.133,A -85,B 0,C 180,E1 -27673.134,E2 -27673.134} C_VEL
LIN {X 0,Y 114.773,Z 529.588,A -85,B 0,C 180,E1 -27675.384,E2 -27675.384} C_VEL
LIN {X 0,Y 117.814,Z 517.374,A -85,B 0,C 180,E1 -27676.955,E2 -27676.955} C_VEL
LIN {X 0,Y 120.041,Z 504.404,A -85,B 0,C 180,E1 -27678.06,E2 -27678.06} C_VEL
LIN {X 0,Y 122.331,Z 480.215,A -85,B 0,C 180,E1 -27679.194,E2 -27679.194} C_VEL
LIN {X 0,Y 123.116,Z 470.52,A -85,B 0,C 180,E1 -27679.642,E2 -27679.642} C_VEL
LIN {X 0,Y 119.758,Z 463.093,A -85,B 0,C 180,E1 -27682.795,E2 -27682.795} C_VEL
LIN {X 0,Y 116.045,Z 455.805,A -85,B 0,C 180,E1 -27686.769,E2 -27686.769} C_VEL
LIN {X 0,Y 112.425,Z 449.507,A -85,B 0,C 180,E1 -27691.392,E2 -27691.392} C_VEL
LIN {X 0,Y 109.686,Z 445.373,A -85,B 0,C 180,E1 -27695.687,E2 -27695.687} C_VEL
LIN {X 0,Y 107.319,Z 441.596,A -85,B 0,C 180,E1 -27700.637,E2 -27700.637} C_VEL
LIN {X 0,Y 104.809,Z 437.922,A -85,B 0,C 180,E1 -27709.861,E2 -27709.861} C_VEL
LIN {X 0,Y 104.645,Z 436.223,A -85,B 0,C 180,E1 -27713.029,E2 -27713.029} C_VEL
LIN {X 0,Y 104.734,Z 436.108,A -85,B 0,C 180,E1 -27718.243,E2 -27718.243} C_VEL
LIN {X 0,Y 105.476,Z 439.151,A -85,B 0,C 180,E1 -27724.113,E2 -27724.113} C_VEL
LIN {X 0,Y 107.348,Z 441.35,A -85,B 0,C 180,E1 -27729.716,E2 -27729.716} C_VEL
LIN {X 0,Y 109.249,Z 444.791,A -85,B 0,C 180,E1 -27733.888,E2 -27733.888} C_VEL
LIN {X 0,Y 110.36,Z 446.364,A -85,B 0,C 180,E1 -27735.821,E2 -27735.821} C_VEL
LIN {X 0,Y 113.054,Z 450.746,A -85,B 0,C 180,E1 -27739.874,E2 -27739.874} C_VEL
LIN {X 0,Y 116.281,Z 456.199,A -85,B 0,C 180,E1 -27743.854,E2 -27743.854} C_VEL
LIN {X 0,Y 118.4,Z 460.483,A -85,B 0,C 180,E1 -27746.197,E2 -27746.197} C_VEL
LIN {X 0,Y 121.585,Z 470.196,A -85,B 0,C 180,E1 -27749.649,E2 -27749.649} C_VEL
LIN {X 0,Y 122.76,Z 475.125,A -85,B 0,C 180,E1 -27750.938,E2 -27750.938} C_VEL
LIN {X 0,Y 122.295,Z 482.999,A -85,B 0,C 180,E1 -27751.414,E2 -27751.414} C_VEL
LIN {X 0,Y 119.649,Z 510.708,A -85,B 0,C 180,E1 -27752.641,E2 -27752.641} C_VEL
LIN {X 0,Y 117.176,Z 524.202,A -85,B 0,C 180,E1 -27753.677,E2 -27753.677} C_VEL
LIN {X 0,Y 113.921,Z 536.575,A -85,B 0,C 180,E1 -27755.175,E2 -27755.175} C_VEL
LIN {X 0,Y 109.325,Z 549.213,A -85,B 0,C 180,E1 -27757.296,E2 -27757.296} C_VEL
LIN {X 0,Y 104.435,Z 560.508,A -85,B 0,C 180,E1 -27760.051,E2 -27760.051} C_VEL
LIN {X 0,Y 99.725,Z 569.62,A -85,B 0,C 180,E1 -27763.017,E2 -27763.017} C_VEL
LIN {X 0,Y 94.871,Z 578.136,A -85,B 0,C 180,E1 -27766.747,E2 -27766.747} C_VEL
LIN {X 0,Y 89.584,Z 586.496,A -85,B 0,C 180,E1 -27771.674,E2 -27771.674} C_VEL
LIN {X 0,Y 85.126,Z 593.655,A -85,B 0,C 180,E1 -27777.546,E2 -27777.546} C_VEL
LIN {X 0,Y 81.26,Z 599.815,A -85,B 0,C 180,E1 -27784.378,E2 -27784.378} C_VEL
LIN {X 0,Y 78.591,Z 604.688,A -85,B 0,C 180,E1 -27791.761,E2 -27791.761} C_VEL
LIN {X 0,Y 77.218,Z 608.42,A -85,B 0,C 180,E1 -27799.512,E2 -27799.512} C_VEL
LIN {X 0,Y 76.964,Z 610.34,A -85,B 0,C 180,E1 -27804.761,E2 -27804.761} C_VEL
LIN {X 0,Y 77.106,Z 611.796,A -85,B 0,C 180,E1 -27810,E2 -27810} C_VEL
LIN {X 0,Y 76.963,Z 612.771,A -85,B 0,C 180,E1 -27815.239,E2 -27815.239} C_VEL
LIN {X 0,Y 78.04,Z 613.551,A -85,B 0,C 180,E1 -27825.674,E2 -27825.674} C_VEL
LIN {X 0,Y 79.462,Z 613.357,A -85,B 0,C 180,E1 -27830.718,E2 -27830.718} C_VEL
LIN {X 0,Y 84.091,Z 611.76,A -85,B 0,C 180,E1 -27840.096,E2 -27840.096} C_VEL
LIN {X 0,Y 87.212,Z 610.387,A -85,B 0,C 180,E1 -27844.339,E2 -27844.339} C_VEL
LIN {X 0,Y 92.734,Z 607.524,A -85,B 0,C 180,E1 -27850.103,E2 -27850.103} C_VEL
LIN {X 0,Y 99.005,Z 603.656,A -85,B 0,C 180,E1 -27855.222,E2 -27855.222} C_VEL
LIN {X 0,Y 106.01,Z 598.69,A -85,B 0,C 180,E1 -27859.675,E2 -27859.675} C_VEL
LIN {X 0,Y 113.683,Z 592.475,A -85,B 0,C 180,E1 -27863.48,E2 -27863.48} C_VEL
LIN {X 0,Y 121.859,Z 584.762,A -85,B 0,C 180,E1 -27866.746,E2 -27866.746} C_VEL
LIN {X 0,Y 130.368,Z 575.114,A -85,B 0,C 180,E1 -27869.601,E2 -27869.601} C_VEL
LIN {X 0,Y 137.795,Z 565.174,A -85,B 0,C 180,E1 -27871.616,E2 -27871.616} C_VEL
LIN {X 0,Y 144.579,Z 553.982,A -85,B 0,C 180,E1 -27873.276,E2 -27873.276} C_VEL
LIN {X 0,Y 149.974,Z 543.032,A -85,B 0,C 180,E1 -27874.43,E2 -27874.43} C_VEL
LIN {X 0,Y 154.64,Z 530.93,A -85,B 0,C 180,E1 -27875.358,E2 -27875.358} C_VEL
LIN {X 0,Y 158.219,Z 518.131,A -85,B 0,C 180,E1 -27876.033,E2 -27876.033} C_VEL
LIN {X 0,Y 160.261,Z 506.697,A -85,B 0,C 180,E1 -27876.496,E2 -27876.496} C_VEL
LIN {X 0,Y 158.72,Z 500.629,A -85,B 0,C 180,E1 -27879.144,E2 -27879.144} C_VEL
LIN {X 0,Y 156.896,Z 494.597,A -85,B 0,C 180,E1 -27882.653,E2 -27882.653} C_VEL
LIN {X 0,Y 155.904,Z 491.674,A -85,B 0,C 180,E1 -27884.978,E2 -27884.978} C_VEL
LIN {X 0,Y 154.881,Z 489.311,A -85,B 0,C 180,E1 -27887.886,E2 -27887.886} C_VEL
LIN {X 0,Y 154.465,Z 488.723,A -85,B 0,C 180,E1 -27889.293,E2 -27889.293} C_VEL
LIN {X 0,Y 153.938,Z 488.386,A -85,B 0,C 180,E1 -27891.478,E2 -27891.478} C_VEL
LIN {X 0,Y 153.487,Z 489.27,A -85,B 0,C 180,E1 -27893.669,E2 -27893.669} C_VEL
LIN {X 0,Y 153.299,Z 494.912,A -85,B 0,C 180,E1 -27900.966,E2 -27900.966} C_VEL
LIN {X 0,Y 154.032,Z 496.434,A -85,B 0,C 180,E1 -27903.902,E2 -27903.902} C_VEL
LIN {X 0,Y 155.492,Z 500.169,A -85,B 0,C 180,E1 -27907.957,E2 -27907.957} C_VEL
LIN {X 0,Y 157.042,Z 504.15,A -85,B 0,C 180,E1 -27911.223,E2 -27911.223} C_VEL
LIN {X 0,Y 157.791,Z 506.406,A -85,B 0,C 180,E1 -27912.746,E2 -27912.746} C_VEL
LIN {X 0,Y 154.976,Z 519.174,A -85,B 0,C 180,E1 -27913.362,E2 -27913.362} C_VEL
LIN {X 0,Y 150.947,Z 531.696,A -85,B 0,C 180,E1 -27914.304,E2 -27914.304} C_VEL
LIN {X 0,Y 145.784,Z 543.446,A -85,B 0,C 180,E1 -27915.39,E2 -27915.39} C_VEL
LIN {X 0,Y 140.286,Z 553.452,A -85,B 0,C 180,E1 -27916.645,E2 -27916.645} C_VEL
LIN {X 0,Y 133.426,Z 563.887,A -85,B 0,C 180,E1 -27918.541,E2 -27918.541} C_VEL
LIN {X 0,Y 125.95,Z 573.191,A -85,B 0,C 180,E1 -27920.833,E2 -27920.833} C_VEL
LIN {X 0,Y 117.193,Z 582.186,A -85,B 0,C 180,E1 -27923.863,E2 -27923.863} C_VEL
LIN {X 0,Y 108.851,Z 589.379,A -85,B 0,C 180,E1 -27927.408,E2 -27927.408} C_VEL
LIN {X 0,Y 102.223,Z 594.204,A -85,B 0,C 180,E1 -27930.753,E2 -27930.753} C_VEL
LIN {X 0,Y 94.778,Z 598.853,A -85,B 0,C 180,E1 -27935.348,E2 -27935.348} C_VEL
LIN {X 0,Y 90.163,Z 601.302,A -85,B 0,C 180,E1 -27938.789,E2 -27938.789} C_VEL
LIN {X 0,Y 85.902,Z 603.279,A -85,B 0,C 180,E1 -27942.582,E2 -27942.582} C_VEL
LIN {X 0,Y 82.036,Z 604.832,A -85,B 0,C 180,E1 -27946.738,E2 -27946.738} C_VEL
LIN {X 0,Y 78.655,Z 605.949,A -85,B 0,C 180,E1 -27951.285,E2 -27951.285} C_VEL
LIN {X 0,Y 73.385,Z 606.91,A -85,B 0,C 180,E1 -27961.391,E2 -27961.391} C_VEL
LIN {X 0,Y 71.581,Z 606.809,A -85,B 0,C 180,E1 -27966.876,E2 -27966.876} C_VEL
LIN {X 0,Y 70.375,Z 606.289,A -85,B 0,C 180,E1 -27972.567,E2 -27972.567} C_VEL
LIN {X 0,Y 69.876,Z 604.011,A -85,B 0,C 180,E1 -27984.228,E2 -27984.228} C_VEL
LIN {X 0,Y 70.91,Z 601.221,A -85,B 0,C 180,E1 -27992.84,E2 -27992.84} C_VEL
LIN {X 0,Y 72.916,Z 597.443,A -85,B 0,C 180,E1 -28001.114,E2 -28001.114} C_VEL
LIN {X 0,Y 76.3,Z 592.539,A -85,B 0,C 180,E1 -28008.807,E2 -28008.807} C_VEL
LIN {X 0,Y 80.724,Z 586.379,A -85,B 0,C 180,E1 -28015.804,E2 -28015.804} C_VEL
LIN {X 0,Y 86.084,Z 578.716,A -85,B 0,C 180,E1 -28022.05,E2 -28022.05} C_VEL
LIN {X 0,Y 92.335,Z 569.087,A -85,B 0,C 180,E1 -28027.51,E2 -28027.51} C_VEL
LIN {X 0,Y 98.132,Z 559.138,A -85,B 0,C 180,E1 -28031.487,E2 -28031.487} C_VEL
LIN {X 0,Y 103.019,Z 549.307,A -85,B 0,C 180,E1 -28034.366,E2 -28034.366} C_VEL
LIN {X 0,Y 107.347,Z 538.665,A -85,B 0,C 180,E1 -28036.747,E2 -28036.747} C_VEL
LIN {X 0,Y 111.506,Z 525.862,A -85,B 0,C 180,E1 -28038.797,E2 -28038.797} C_VEL
LIN {X 0,Y 114.418,Z 513.612,A -85,B 0,C 180,E1 -28040.175,E2 -28040.175} C_VEL
LIN {X 0,Y 116.409,Z 500.576,A -85,B 0,C 180,E1 -28041.106,E2 -28041.106} C_VEL
LIN {X 0,Y 118.89,Z 473.239,A -85,B 0,C 180,E1 -28042.329,E2 -28042.329} C_VEL
LIN {X 0,Y 114.985,Z 464.493,A -85,B 0,C 180,E1 -28046.625,E2 -28046.625} C_VEL
LIN {X 0,Y 111.709,Z 458.204,A -85,B 0,C 180,E1 -28050.864,E2 -28050.864} C_VEL
LIN {X 0,Y 109.729,Z 454.811,A -85,B 0,C 180,E1 -28053.874,E2 -28053.874} C_VEL
LIN {X 0,Y 107.989,Z 451.827,A -85,B 0,C 180,E1 -28057.014,E2 -28057.014} C_VEL
LIN {X 0,Y 105.654,Z 447.883,A -85,B 0,C 180,E1 -28062.581,E2 -28062.581} C_VEL
LIN {X 0,Y 103.892,Z 445.116,A -85,B 0,C 180,E1 -28070.017,E2 -28070.017} C_VEL
LIN {X 0,Y 103.742,Z 443.219,A -85,B 0,C 180,E1 -28073.723,E2 -28073.723} C_VEL
LIN {X 0,Y 103.805,Z 443.167,A -85,B 0,C 180,E1 -28077.574,E2 -28077.574} C_VEL
LIN {X 0,Y 104.632,Z 446.418,A -85,B 0,C 180,E1 -28084.333,E2 -28084.333} C_VEL
LIN {X 0,Y 105.972,Z 448.048,A -85,B 0,C 180,E1 -28088.578,E2 -28088.578} C_VEL
LIN {X 0,Y 108.057,Z 451.834,A -85,B 0,C 180,E1 -28093.452,E2 -28093.452} C_VEL
LIN {X 0,Y 110.939,Z 456.858,A -85,B 0,C 180,E1 -28098.376,E2 -28098.376} C_VEL
LIN {X 0,Y 113.843,Z 462.195,A -85,B 0,C 180,E1 -28102.336,E2 -28102.336} C_VEL
LIN {X 0,Y 115.415,Z 465.569,A -85,B 0,C 180,E1 -28104.264,E2 -28104.264} C_VEL
LIN {X 0,Y 118.27,Z 475.257,A -85,B 0,C 180,E1 -28107.781,E2 -28107.781} C_VEL
LIN {X 0,Y 118.715,Z 477.218,A -85,B 0,C 180,E1 -28108.334,E2 -28108.334} C_VEL
LIN {X 0,Y 115.591,Z 510.007,A -85,B 0,C 180,E1 -28109.808,E2 -28109.808} C_VEL
LIN {X 0,Y 113.018,Z 523.564,A -85,B 0,C 180,E1 -28110.806,E2 -28110.806} C_VEL
LIN {X 0,Y 109.615,Z 536.039,A -85,B 0,C 180,E1 -28112.275,E2 -28112.275} C_VEL
LIN {X 0,Y 105.153,Z 547.927,A -85,B 0,C 180,E1 -28114.201,E2 -28114.201} C_VEL
LIN {X 0,Y 100.004,Z 559.4,A -85,B 0,C 180,E1 -28116.929,E2 -28116.929} C_VEL
LIN {X 0,Y 94.943,Z 568.631,A -85,B 0,C 180,E1 -28119.828,E2 -28119.828} C_VEL
LIN {X 0,Y 89.793,Z 577.271,A -85,B 0,C 180,E1 -28123.617,E2 -28123.617} C_VEL
LIN {X 0,Y 84.513,Z 585.218,A -85,B 0,C 180,E1 -28128.298,E2 -28128.298} C_VEL
LIN {X 0,Y 80.884,Z 590.572,A -85,B 0,C 180,E1 -28132.54,E2 -28132.54} C_VEL
LIN {X 0,Y 76.229,Z 597.296,A -85,B 0,C 180,E1 -28139.531,E2 -28139.531} C_VEL
LIN {X 0,Y 72.665,Z 602.639,A -85,B 0,C 180,E1 -28147.241,E2 -28147.241} C_VEL
LIN {X 0,Y 70.608,Z 606.798,A -85,B 0,C 180,E1 -28155.592,E2 -28155.592} C_VEL
LIN {X 0,Y 69.883,Z 609.872,A -85,B 0,C 180,E1 -28164.228,E2 -28164.228} C_VEL
LIN {X 0,Y 70.022,Z 611.377,A -85,B 0,C 180,E1 -28170,E2 -28170} C_VEL
LIN {X 0,Y 69.883,Z 612.377,A -85,B 0,C 180,E1 -28175.772,E2 -28175.772} C_VEL
LIN {X 0,Y 71.2,Z 613.204,A -85,B 0,C 180,E1 -28187.225,E2 -28187.225} C_VEL
LIN {X 0,Y 72.838,Z 613.047,A -85,B 0,C 180,E1 -28192.702,E2 -28192.702} C_VEL
LIN {X 0,Y 75.078,Z 612.471,A -85,B 0,C 180,E1 -28197.907,E2 -28197.907} C_VEL
LIN {X 0,Y 81.423,Z 610.16,A -85,B 0,C 180,E1 -28207.17,E2 -28207.17} C_VEL
LIN {X 0,Y 87.383,Z 607.347,A -85,B 0,C 180,E1 -28213.127,E2 -28213.127} C_VEL
LIN {X 0,Y 94.122,Z 603.534,A -85,B 0,C 180,E1 -28218.303,E2 -28218.303} C_VEL
LIN {X 0,Y 101.556,Z 598.625,A -85,B 0,C 180,E1 -28222.733,E2 -28222.733} C_VEL
LIN {X 0,Y 109.602,Z 592.474,A -85,B 0,C 180,E1 -28226.468,E2 -28226.468} C_VEL
LIN {X 0,Y 118.118,Z 584.856,A -85,B 0,C 180,E1 -28229.624,E2 -28229.624} C_VEL
LIN {X 0,Y 126.937,Z 575.311,A -85,B 0,C 180,E1 -28232.355,E2 -28232.355} C_VEL
LIN {X 0,Y 134.576,Z 565.477,A -85,B 0,C 180,E1 -28234.267,E2 -28234.267} C_VEL
LIN {X 0,Y 141.544,Z 554.497,A -85,B 0,C 180,E1 -28235.831,E2 -28235.831} C_VEL
LIN {X 0,Y 147.054,Z 543.753,A -85,B 0,C 180,E1 -28236.922,E2 -28236.922} C_VEL
LIN {X 0,Y 152.177,Z 530.955,A -85,B 0,C 180,E1 -28237.846,E2 -28237.846} C_VEL
LIN {X 0,Y 155.764,Z 518.717,A -85,B 0,C 180,E1 -28238.452,E2 -28238.452} C_VEL
LIN {X 0,Y 157.502,Z 509.916,A -85,B 0,C 180,E1 -28238.821,E2 -28238.821} C_VEL
LIN {X 0,Y 156.255,Z 504.1,A -85,B 0,C 180,E1 -28241.73,E2 -28241.73} C_VEL
LIN {X 0,Y 155.119,Z 499.86,A -85,B 0,C 180,E1 -28244.521,E2 -28244.521} C_VEL
LIN {X 0,Y 154.574,Z 498.12,A -85,B 0,C 180,E1 -28246.023,E2 -28246.023} C_VEL
LIN {X 0,Y 153.812,Z 496.179,A -85,B 0,C 180,E1 -28248.469,E2 -28248.469} C_VEL
LIN {X 0,Y 152.929,Z 493.074,A -85,B 0,C 180,E1 -28254.727,E2 -28254.727} C_VEL
LIN {X 0,Y 152.963,Z 493.22,A -85,B 0,C 180,E1 -28257.697,E2 -28257.697} C_VEL
LIN {X 0,Y 153.299,Z 494.912,A -85,B 0,C 180,E1 -28260.966,E2 -28260.966} C_VEL
LIN {X 0,Y 153.499,Z 496.368,A -85,B 0,C 180,E1 -28262.33,E2 -28262.33} C_VEL
LIN {X 0,Y 153.623,Z 500.577,A -85,B 0,C 180,E1 -28264.267,E2 -28264.267} C_VEL
LIN {X 0,Y 153.749,Z 505.139,A -85,B 0,C 180,E1 -28266.163,E2 -28266.163} C_VEL
LIN {X 0,Y 154.025,Z 507.125,A -85,B 0,C 180,E1 -28267.471,E2 -28267.471} C_VEL
LIN {X 0,Y 155.07,Z 510.58,A -85,B 0,C 180,E1 -28270.363,E2 -28270.363} C_VEL
LIN {X 0,Y 152.098,Z 522.399,A -85,B 0,C 180,E1 -28271.026,E2 -28271.026} C_VEL
LIN {X 0,Y 147.706,Z 534.773,A -85,B 0,C 180,E1 -28271.941,E2 -28271.941} C_VEL
LIN {X 0,Y 142.409,Z 545.94,A -85,B 0,C 180,E1 -28272.927,E2 -28272.927} C_VEL
LIN {X 0,Y 135.833,Z 556.977,A -85,B 0,C 180,E1 -28274.349,E2 -28274.349} C_VEL
LIN {X 0,Y 128.056,Z 567.733,A -85,B 0,C 180,E1 -28276.434,E2 -28276.434} C_VEL
LIN {X 0,Y 120.501,Z 576.273,A -85,B 0,C 180,E1 -28278.607,E2 -28278.607} C_VEL
LIN {X 0,Y 111.491,Z 584.679,A -85,B 0,C 180,E1 -28281.604,E2 -28281.604} C_VEL
LIN {X 0,Y 102.87,Z 591.409,A -85,B 0,C 180,E1 -28285.149,E2 -28285.149} C_VEL
LIN {X 0,Y 93.366,Z 597.527,A -85,B 0,C 180,E1 -28290.045,E2 -28290.045} C_VEL
LIN {X 0,Y 85.81,Z 601.462,A -85,B 0,C 180,E1 -28295.016,E2 -28295.016} C_VEL
LIN {X 0,Y 81.177,Z 603.468,A -85,B 0,C 180,E1 -28298.815,E2 -28298.815} C_VEL
LIN {X 0,Y 76.909,Z 605.049,A -85,B 0,C 180,E1 -28303.028,E2 -28303.028} C_VEL
LIN {X 0,Y 73.131,Z 606.214,A -85,B 0,C 180,E1 -28307.725,E2 -28307.725} C_VEL
LIN {X 0,Y 67.135,Z 607.236,A -85,B 0,C 180,E1 -28318.439,E2 -28318.439} C_VEL
LIN {X 0,Y 64.997,Z 607.162,A -85,B 0,C 180,E1 -28324.374,E2 -28324.374} C_VEL
LIN {X 0,Y 63.528,Z 606.692,A -85,B 0,C 180,E1 -28330.617,E2 -28330.617} C_VEL
LIN {X 0,Y 62.775,Z 605.779,A -85,B 0,C 180,E1 -28337.062,E2 -28337.062} C_VEL
LIN {X 0,Y 63.266,Z 603.076,A -85,B 0,C 180,E1 -28348.892,E2 -28348.892} C_VEL
LIN {X 0,Y 65.121,Z 599.38,A -85,B 0,C 180,E1 -28359.316,E2 -28359.316} C_VEL
LIN {X 0,Y 68.262,Z 594.932,A -85,B 0,C 180,E1 -28367.991,E2 -28367.991} C_VEL
LIN {X 0,Y 73.538,Z 588.195,A -85,B 0,C 180,E1 -28376.997,E2 -28376.997} C_VEL
LIN {X 0,Y 79.152,Z 580.874,A -85,B 0,C 180,E1 -28383.706,E2 -28383.706} C_VEL
LIN {X 0,Y 85.694,Z 571.776,A -85,B 0,C 180,E1 -28389.464,E2 -28389.464} C_VEL
LIN {X 0,Y 92.343,Z 561.244,A -85,B 0,C 180,E1 -28393.985,E2 -28393.985} C_VEL
LIN {X 0,Y 98.101,Z 550.527,A -85,B 0,C 180,E1 -28397.248,E2 -28397.248} C_VEL
LIN {X 0,Y 102.646,Z 540.152,A -85,B 0,C 180,E1 -28399.613,E2 -28399.613} C_VEL
LIN {X 0,Y 107.016,Z 527.678,A -85,B 0,C 180,E1 -28401.624,E2 -28401.624} C_VEL
LIN {X 0,Y 110.408,Z 514.385,A -85,B 0,C 180,E1 -28403.137,E2 -28403.137} C_VEL
LIN {X 0,Y 112.485,Z 501.766,A -85,B 0,C 180,E1 -28404.05,E2 -28404.05} C_VEL
LIN {X 0,Y 114.931,Z 476.231,A -85,B 0,C 180,E1 -28405.186,E2 -28405.186} C_VEL
LIN {X 0,Y 111.793,Z 468.93,A -85,B 0,C 180,E1 -28409.17,E2 -28409.17} C_VEL
LIN {X 0,Y 109.173,Z 463.486,A -85,B 0,C 180,E1 -28413.086,E2 -28413.086} C_VEL
LIN {X 0,Y 107.472,Z 460.364,A -85,B 0,C 180,E1 -28416.073,E2 -28416.073} C_VEL
LIN {X 0,Y 106.328,Z 458.279,A -85,B 0,C 180,E1 -28418.427,E2 -28418.427} C_VEL
LIN {X 0,Y 104.424,Z 454.713,A -85,B 0,C 180,E1 -28423.521,E2 -28423.521} C_VEL
LIN {X 0,Y 102.889,Z 451.794,A -85,B 0,C 180,E1 -28431.263,E2 -28431.263} C_VEL
LIN {X 0,Y 102.854,Z 450.253,A -85,B 0,C 180,E1 -28434.273,E2 -28434.273} C_VEL
LIN {X 0,Y 102.893,Z 450.403,A -85,B 0,C 180,E1 -28437.307,E2 -28437.307} C_VEL
LIN {X 0,Y 103.802,Z 453.706,A -85,B 0,C 180,E1 -28444.611,E2 -28444.611} C_VEL
LIN {X 0,Y 104.658,Z 454.799,A -85,B 0,C 180,E1 -28447.475,E2 -28447.475} C_VEL
LIN {X 0,Y 107.032,Z 459.505,A -85,B 0,C 180,E1 -28453.406,E2 -28453.406} C_VEL
LIN {X 0,Y 108.931,Z 463.071,A -85,B 0,C 180,E1 -28456.877,E2 -28456.877} C_VEL
LIN {X 0,Y 111.278,Z 467.647,A -85,B 0,C 180,E1 -28460.446,E2 -28460.446} C_VEL
LIN {X 0,Y 112.644,Z 470.933,A -85,B 0,C 180,E1 -28462.345,E2 -28462.345} C_VEL
LIN {X 0,Y 114.853,Z 479.393,A -85,B 0,C 180,E1 -28465.494,E2 -28465.494} C_VEL
LIN {X 0,Y 111.682,Z 510.26,A -85,B 0,C 180,E1 -28466.829,E2 -28466.829} C_VEL
LIN {X 0,Y 108.986,Z 523.696,A -85,B 0,C 180,E1 -28467.793,E2 -28467.793} C_VEL
LIN {X 0,Y 105.267,Z 536.519,A -85,B 0,C 180,E1 -28469.299,E2 -28469.299} C_VEL
LIN {X 0,Y 100.614,Z 548.235,A -85,B 0,C 180,E1 -28471.168,E2 -28471.168} C_VEL
LIN {X 0,Y 95.213,Z 559.591,A -85,B 0,C 180,E1 -28473.862,E2 -28473.862} C_VEL
LIN {X 0,Y 89.896,Z 568.733,A -85,B 0,C 180,E1 -28476.744,E2 -28476.744} C_VEL
LIN {X 0,Y 83.839,Z 578.143,A -85,B 0,C 180,E1 -28481.024,E2 -28481.024} C_VEL
LIN {X 0,Y 77.753,Z 586.45,A -85,B 0,C 180,E1 -28486.31,E2 -28486.31} C_VEL
LIN {X 0,Y 72.566,Z 593.443,A -85,B 0,C 180,E1 -28492.75,E2 -28492.75} C_VEL
LIN {X 0,Y 68.682,Z 598.603,A -85,B 0,C 180,E1 -28499.228,E2 -28499.228} C_VEL
LIN {X 0,Y 65.153,Z 603.587,A -85,B 0,C 180,E1 -28507.819,E2 -28507.819} C_VEL
LIN {X 0,Y 63.253,Z 607.431,A -85,B 0,C 180,E1 -28517.161,E2 -28517.161} C_VEL
LIN {X 0,Y 62.799,Z 609.403,A -85,B 0,C 180,E1 -28523.575,E2 -28523.575} C_VEL
LIN {X 0,Y 62.925,Z 610.947,A -85,B 0,C 180,E1 -28530,E2 -28530} C_VEL
LIN {X 0,Y 62.815,Z 611.983,A -85,B 0,C 180,E1 -28536.424,E2 -28536.424} C_VEL
LIN {X 0,Y 64.433,Z 612.857,A -85,B 0,C 180,E1 -28549.1,E2 -28549.1} C_VEL
LIN {X 0,Y 66.303,Z 612.726,A -85,B 0,C 180,E1 -28555.086,E2 -28555.086} C_VEL
LIN {X 0,Y 68.863,Z 612.195,A -85,B 0,C 180,E1 -28560.682,E2 -28560.682} C_VEL
LIN {X 0,Y 75.866,Z 609.934,A -85,B 0,C 180,E1 -28570.424,E2 -28570.424} C_VEL
LIN {X 0,Y 83.281,Z 606.71,A -85,B 0,C 180,E1 -28577.325,E2 -28577.325} C_VEL
LIN {X 0,Y 92.093,Z 601.944,A -85,B 0,C 180,E1 -28583.252,E2 -28583.252} C_VEL
LIN {X 0,Y 101.554,Z 595.683,A -85,B 0,C 180,E1 -28587.966,E2 -28587.966} C_VEL
LIN {X 0,Y 110.235,Z 588.901,A -85,B 0,C 180,E1 -28591.235,E2 -28591.235} C_VEL
LIN {X 0,Y 119.229,Z 580.507,A -85,B 0,C 180,E1 -28594.013,E2 -28594.013} C_VEL
LIN {X 0,Y 126.937,Z 571.882,A -85,B 0,C 180,E1 -28595.996,E2 -28595.996} C_VEL
LIN {X 0,Y 134.017,Z 562.452,A -85,B 0,C 180,E1 -28597.555,E2 -28597.555} C_VEL
LIN {X 0,Y 141.21,Z 550.772,A -85,B 0,C 180,E1 -28598.933,E2 -28598.933} C_VEL
LIN {X 0,Y 146.887,Z 539.138,A -85,B 0,C 180,E1 -28599.878,E2 -28599.878} C_VEL
LIN {X 0,Y 151.577,Z 526.292,A -85,B 0,C 180,E1 -28600.662,E2 -28600.662} C_VEL
LIN {X 0,Y 154.785,Z 514.043,A -85,B 0,C 180,E1 -28601.147,E2 -28601.147} C_VEL
LIN {X 0,Y 154.886,Z 513.152,A -85,B 0,C 180,E1 -28601.31,E2 -28601.31} C_VEL
LIN {X 0,Y 153.952,Z 507.503,A -85,B 0,C 180,E1 -28604.592,E2 -28604.592} C_VEL
LIN {X 0,Y 153.273,Z 504.696,A -85,B 0,C 180,E1 -28606.915,E2 -28606.915} C_VEL
LIN {X 0,Y 152.712,Z 503.056,A -85,B 0,C 180,E1 -28609.057,E2 -28609.057} C_VEL
LIN {X 0,Y 152.04,Z 500.284,A -85,B 0,C 180,E1 -28614.696,E2 -28614.696} C_VEL
LIN {X 0,Y 152.062,Z 500.41,A -85,B 0,C 180,E1 -28617.683,E2 -28617.683} C_VEL
LIN {X 0,Y 152.859,Z 503.289,A -85,B 0,C 180,E1 -28623.295,E2 -28623.295} C_VEL
LIN {X 0,Y 153.944,Z 506.827,A -85,B 0,C 180,E1 -28627.213,E2 -28627.213} C_VEL
LIN {X 0,Y 154.025,Z 507.125,A -85,B 0,C 180,E1 -28627.471,E2 -28627.471} C_VEL
LIN {X 0,Y 154.128,Z 508.837,A -85,B 0,C 180,E1 -28628.249,E2 -28628.249} C_VEL
LIN {X 0,Y 153.712,Z 511.978,A -85,B 0,C 180,E1 -28628.781,E2 -28628.781} C_VEL
LIN {X 0,Y 152.812,Z 515.798,A -85,B 0,C 180,E1 -28628.937,E2 -28628.937} C_VEL
LIN {X 0,Y 149.301,Z 526.09,A -85,B 0,C 180,E1 -28628.65,E2 -28628.65} C_VEL
LIN {X 0,Y 148.784,Z 527.502,A -85,B 0,C 180,E1 -28628.726,E2 -28628.726} C_VEL
LIN {X 0,Y 144.107,Z 538.998,A -85,B 0,C 180,E1 -28629.571,E2 -28629.571} C_VEL
LIN {X 0,Y 138.482,Z 549.687,A -85,B 0,C 180,E1 -28630.497,E2 -28630.497} C_VEL
LIN {X 0,Y 131.956,Z 559.879,A -85,B 0,C 180,E1 -28631.865,E2 -28631.865} C_VEL
LIN {X 0,Y 124.5,Z 569.481,A -85,B 0,C 180,E1 -28633.716,E2 -28633.716} C_VEL
LIN {X 0,Y 115.246,Z 579.136,A -85,B 0,C 180,E1 -28636.167,E2 -28636.167} C_VEL
LIN {X 0,Y 105.833,Z 587.197,A -85,B 0,C 180,E1 -28639.161,E2 -28639.161} C_VEL
LIN {X 0,Y 98.539,Z 592.431,A -85,B 0,C 180,E1 -28642.003,E2 -28642.003} C_VEL
LIN {X 0,Y 89.947,Z 597.624,A -85,B 0,C 180,E1 -28646.035,E2 -28646.035} C_VEL
LIN {X 0,Y 81.313,Z 601.854,A -85,B 0,C 180,E1 -28651.239,E2 -28651.239} C_VEL
LIN {X 0,Y 72.152,Z 605.269,A -85,B 0,C 180,E1 -28658.811,E2 -28658.811} C_VEL
LIN {X 0,Y 67.929,Z 606.466,A -85,B 0,C 180,E1 -28663.597,E2 -28663.597} C_VEL
LIN {X 0,Y 62.617,Z 607.44,A -85,B 0,C 180,E1 -28671.786,E2 -28671.786} C_VEL
LIN {X 0,Y 58.575,Z 607.515,A -85,B 0,C 180,E1 -28681.32,E2 -28681.32} C_VEL
LIN {X 0,Y 56.77,Z 607.081,A -85,B 0,C 180,E1 -28688.199,E2 -28688.199} C_VEL
LIN {X 0,Y 55.781,Z 606.212,A -85,B 0,C 180,E1 -28695.405,E2 -28695.405} C_VEL
LIN {X 0,Y 56.227,Z 603.336,A -85,B 0,C 180,E1 -28709.638,E2 -28709.638} C_VEL
LIN {X 0,Y 58.141,Z 599.919,A -85,B 0,C 180,E1 -28720.446,E2 -28720.446} C_VEL
LIN {X 0,Y 61.541,Z 595.534,A -85,B 0,C 180,E1 -28730.035,E2 -28730.035} C_VEL
LIN {X 0,Y 66.376,Z 589.957,A -85,B 0,C 180,E1 -28738.454,E2 -28738.454} C_VEL
LIN {X 0,Y 72.329,Z 582.997,A -85,B 0,C 180,E1 -28745.661,E2 -28745.661} C_VEL
LIN {X 0,Y 79.109,Z 574.289,A -85,B 0,C 180,E1 -28751.781,E2 -28751.781} C_VEL
LIN {X 0,Y 85.441,Z 565.347,A -85,B 0,C 180,E1 -28756.031,E2 -28756.031} C_VEL
LIN {X 0,Y 91.421,Z 555.523,A -85,B 0,C 180,E1 -28759.387,E2 -28759.387} C_VEL
LIN {X 0,Y 96.868,Z 544.683,A -85,B 0,C 180,E1 -28762.091,E2 -28762.091} C_VEL
LIN {X 0,Y 101.756,Z 532.549,A -85,B 0,C 180,E1 -28764.245,E2 -28764.245} C_VEL
LIN {X 0,Y 105.271,Z 521.13,A -85,B 0,C 180,E1 -28765.71,E2 -28765.71} C_VEL
LIN {X 0,Y 108.085,Z 508.239,A -85,B 0,C 180,E1 -28766.846,E2 -28766.846} C_VEL
LIN {X 0,Y 109.955,Z 493.244,A -85,B 0,C 180,E1 -28767.607,E2 -28767.607} C_VEL
LIN {X 0,Y 111.27,Z 479.326,A -85,B 0,C 180,E1 -28768.228,E2 -28768.228} C_VEL
LIN {X 0,Y 108.723,Z 472.957,A -85,B 0,C 180,E1 -28772.052,E2 -28772.052} C_VEL
LIN {X 0,Y 106.37,Z 467.841,A -85,B 0,C 180,E1 -28776.27,E2 -28776.27} C_VEL
LIN {X 0,Y 104.737,Z 464.698,A -85,B 0,C 180,E1 -28779.884,E2 -28779.884} C_VEL
LIN {X 0,Y 103.163,Z 461.466,A -85,B 0,C 180,E1 -28784.692,E2 -28784.692} C_VEL
LIN {X 0,Y 101.932,Z 458.36,A -85,B 0,C 180,E1 -28792.763,E2 -28792.763} C_VEL
LIN {X 0,Y 101.978,Z 457.268,A -85,B 0,C 180,E1 -28794.832,E2 -28794.832} C_VEL
LIN {X 0,Y 101.995,Z 457.353,A -85,B 0,C 180,E1 -28796.542,E2 -28796.542} C_VEL
LIN {X 0,Y 102.83,Z 460.724,A -85,B 0,C 180,E1 -28804.286,E2 -28804.286} C_VEL
LIN {X 0,Y 103.416,Z 461.621,A -85,B 0,C 180,E1 -28806.462,E2 -28806.462} C_VEL
LIN {X 0,Y 105.395,Z 465.938,A -85,B 0,C 180,E1 -28812.027,E2 -28812.027} C_VEL
LIN {X 0,Y 107.261,Z 469.784,A -85,B 0,C 180,E1 -28815.802,E2 -28815.802} C_VEL
LIN {X 0,Y 109.668,Z 475.147,A -85,B 0,C 180,E1 -28819.781,E2 -28819.781} C_VEL
LIN {X 0,Y 111.217,Z 481.74,A -85,B 0,C 180,E1 -28822.414,E2 -28822.414} C_VEL
LIN {X 0,Y 108.215,Z 509.806,A -85,B 0,C 180,E1 -28823.608,E2 -28823.608} C_VEL
LIN {X 0,Y 105.463,Z 523.092,A -85,B 0,C 180,E1 -28824.503,E2 -28824.503} C_VEL
LIN {X 0,Y 102.257,Z 534.024,A -85,B 0,C 180,E1 -28825.673,E2 -28825.673} C_VEL
LIN {X 0,Y 97.876,Z 545.349,A -85,B 0,C 180,E1 -28827.306,E2 -28827.306} C_VEL
LIN {X 0,Y 92.069,Z 557.156,A -85,B 0,C 180,E1 -28829.741,E2 -28829.741} C_VEL
LIN {X 0,Y 85.838,Z 567.76,A -85,B 0,C 180,E1 -28832.944,E2 -28832.944} C_VEL
LIN {X 0,Y 79.331,Z 577.314,A -85,B 0,C 180,E1 -28837.127,E2 -28837.127} C_VEL
LIN {X 0,Y 73.306,Z 585.082,A -85,B 0,C 180,E1 -28841.956,E2 -28841.956} C_VEL
LIN {X 0,Y 69.952,Z 589.143,A -85,B 0,C 180,E1 -28845.31,E2 -28845.31} C_VEL
LIN {X 0,Y 65.152,Z 594.991,A -85,B 0,C 180,E1 -28851.666,E2 -28851.666} C_VEL
LIN {X 0,Y 61.111,Z 599.827,A -85,B 0,C 180,E1 -28858.835,E2 -28858.835} C_VEL
LIN {X 0,Y 57.639,Z 604.48,A -85,B 0,C 180,E1 -28868.544,E2 -28868.544} C_VEL
LIN {X 0,Y 55.913,Z 608.012,A -85,B 0,C 180,E1 -28879.132,E2 -28879.132} C_VEL
LIN {X 0,Y 55.821,Z 610.506,A -85,B 0,C 180,E1 -28890,E2 -28890} C_VEL
LIN {X 0,Y 55.759,Z 611.589,A -85,B 0,C 180,E1 -28897.241,E2 -28897.241} C_VEL
LIN {X 0,Y 57.756,Z 612.51,A -85,B 0,C 180,E1 -28911.41,E2 -28911.41} C_VEL
LIN {X 0,Y 62.847,Z 611.915,A -85,B 0,C 180,E1 -28923.995,E2 -28923.995} C_VEL
LIN {X 0,Y 70.594,Z 609.707,A -85,B 0,C 180,E1 -28934.177,E2 -28934.177} C_VEL
LIN {X 0,Y 79.324,Z 606.226,A -85,B 0,C 180,E1 -28941.672,E2 -28941.672} C_VEL
LIN {X 0,Y 88.009,Z 601.847,A -85,B 0,C 180,E1 -28946.978,E2 -28946.978} C_VEL
LIN {X 0,Y 97.97,Z 595.66,A -85,B 0,C 180,E1 -28951.491,E2 -28951.491} C_VEL
LIN {X 0,Y 107.004,Z 588.949,A -85,B 0,C 180,E1 -28954.566,E2 -28954.566} C_VEL
LIN {X 0,Y 116.301,Z 580.65,A -85,B 0,C 180,E1 -28957.15,E2 -28957.15} C_VEL
LIN {X 0,Y 124.226,Z 572.15,A -85,B 0,C 180,E1 -28958.98,E2 -28958.98} C_VEL
LIN {X 0,Y 131.481,Z 562.844,A -85,B 0,C 180,E1 -28960.404,E2 -28960.404} C_VEL
LIN {X 0,Y 138.827,Z 551.32,A -85,B 0,C 180,E1 -28961.656,E2 -28961.656} C_VEL
LIN {X 0,Y 144.607,Z 539.975,A -85,B 0,C 180,E1 -28962.509,E2 -28962.509} C_VEL
LIN {X 0,Y 149.035,Z 528.659,A -85,B 0,C 180,E1 -28963.173,E2 -28963.173} C_VEL
LIN {X 0,Y 152.323,Z 517.412,A -85,B 0,C 180,E1 -28963.607,E2 -28963.607} C_VEL
LIN {X 0,Y 152.347,Z 516.339,A -85,B 0,C 180,E1 -28964.018,E2 -28964.018} C_VEL
LIN {X 0,Y 151.89,Z 511.926,A -85,B 0,C 180,E1 -28967.049,E2 -28967.049} C_VEL
LIN {X 0,Y 151.356,Z 509.886,A -85,B 0,C 180,E1 -28969.635,E2 -28969.635} C_VEL
LIN {X 0,Y 150.909,Z 507.452,A -85,B 0,C 180,E1 -28974.656,E2 -28974.656} C_VEL
LIN {X 0,Y 150.905,Z 507.561,A -85,B 0,C 180,E1 -28977.665,E2 -28977.665} C_VEL
LIN {X 0,Y 151.393,Z 510.036,A -85,B 0,C 180,E1 -28982.661,E2 -28982.661} C_VEL
LIN {X 0,Y 152.131,Z 513.568,A -85,B 0,C 180,E1 -28986.633,E2 -28986.633} C_VEL
LIN {X 0,Y 152.486,Z 515.029,A -85,B 0,C 180,E1 -28987.994,E2 -28987.994} C_VEL
LIN {X 0,Y 148.784,Z 527.502,A -85,B 0,C 180,E1 -28988.726,E2 -28988.726} C_VEL
LIN {X 0,Y 146.561,Z 533.082,A -85,B 0,C 180,E1 -28988.881,E2 -28988.881} C_VEL
LIN {X 0,Y 142.006,Z 541.863,A -85,B 0,C 180,E1 -28988.416,E2 -28988.416} C_VEL
LIN {X 0,Y 136.853,Z 550.203,A -85,B 0,C 180,E1 -28987.97,E2 -28987.97} C_VEL
LIN {X 0,Y 133.683,Z 555.048,A -85,B 0,C 180,E1 -28988.196,E2 -28988.196} C_VEL
LIN {X 0,Y 126.86,Z 564.542,A -85,B 0,C 180,E1 -28989.568,E2 -28989.568} C_VEL
LIN {X 0,Y 118.335,Z 574.252,A -85,B 0,C 180,E1 -28991.5,E2 -28991.5} C_VEL
LIN {X 0,Y 108.609,Z 583.233,A -85,B 0,C 180,E1 -28993.924,E2 -28993.924} C_VEL
LIN {X 0,Y 98.795,Z 590.651,A -85,B 0,C 180,E1 -28997.013,E2 -28997.013} C_VEL
LIN {X 0,Y 89.987,Z 596.09,A -85,B 0,C 180,E1 -29000.417,E2 -29000.417} C_VEL
LIN {X 0,Y 81.218,Z 600.525,A -85,B 0,C 180,E1 -29004.692,E2 -29004.692} C_VEL
LIN {X 0,Y 72.959,Z 603.855,A -85,B 0,C 180,E1 -29009.896,E2 -29009.896} C_VEL
LIN {X 0,Y 67.84,Z 605.491,A -85,B 0,C 180,E1 -29014.029,E2 -29014.029} C_VEL
LIN {X 0,Y 63.153,Z 606.714,A -85,B 0,C 180,E1 -29018.833,E2 -29018.833} C_VEL
LIN {X 0,Y 56.555,Z 607.808,A -85,B 0,C 180,E1 -29028.215,E2 -29028.215} C_VEL
LIN {X 0,Y 52.366,Z 607.866,A -85,B 0,C 180,E1 -29037.532,E2 -29037.532} C_VEL
LIN {X 0,Y 50.141,Z 607.459,A -85,B 0,C 180,E1 -29045.135,E2 -29045.135} C_VEL
LIN {X 0,Y 48.859,Z 606.642,A -85,B 0,C 180,E1 -29053.281,E2 -29053.281} C_VEL
LIN {X 0,Y 49.115,Z 603.728,A -85,B 0,C 180,E1 -29070,E2 -29070} C_VEL
LIN {X 0,Y 51.188,Z 600.454,A -85,B 0,C 180,E1 -29081.885,E2 -29081.885} C_VEL
LIN {X 0,Y 54.918,Z 596.131,A -85,B 0,C 180,E1 -29092.576,E2 -29092.576} C_VEL
LIN {X 0,Y 60.246,Z 590.617,A -85,B 0,C 180,E1 -29101.664,E2 -29101.664} C_VEL
LIN {X 0,Y 66.705,Z 583.745,A -85,B 0,C 180,E1 -29109.208,E2 -29109.208} C_VEL
LIN {X 0,Y 73.981,Z 575.148,A -85,B 0,C 180,E1 -29115.436,E2 -29115.436} C_VEL
LIN {X 0,Y 80.696,Z 566.308,A -85,B 0,C 180,E1 -29119.644,E2 -29119.644} C_VEL
LIN {X 0,Y 86.98,Z 556.613,A -85,B 0,C 180,E1 -29122.929,E2 -29122.929} C_VEL
LIN {X 0,Y 92.714,Z 546.002,A -85,B 0,C 180,E1 -29125.521,E2 -29125.521} C_VEL
LIN {X 0,Y 97.806,Z 534.151,A -85,B 0,C 180,E1 -29127.596,E2 -29127.596} C_VEL
LIN {X 0,Y 102.033,Z 521.16,A -85,B 0,C 180,E1 -29129.199,E2 -29129.199} C_VEL
LIN {X 0,Y 104.825,Z 508.88,A -85,B 0,C 180,E1 -29130.23,E2 -29130.23} C_VEL
LIN {X 0,Y 106.807,Z 493.865,A -85,B 0,C 180,E1 -29130.955,E2 -29130.955} C_VEL
LIN {X 0,Y 107.919,Z 482.509,A -85,B 0,C 180,E1 -29131.462,E2 -29131.462} C_VEL
LIN {X 0,Y 105.618,Z 476.457,A -85,B 0,C 180,E1 -29135.686,E2 -29135.686} C_VEL
LIN {X 0,Y 103.965,Z 472.686,A -85,B 0,C 180,E1 -29139.386,E2 -29139.386} C_VEL
LIN {X 0,Y 102.164,Z 468.507,A -85,B 0,C 180,E1 -29145.049,E2 -29145.049} C_VEL
LIN {X 0,Y 101.031,Z 465.335,A -85,B 0,C 180,E1 -29153.394,E2 -29153.394} C_VEL
LIN {X 0,Y 101.102,Z 464.362,A -85,B 0,C 180,E1 -29155.4,E2 -29155.4} C_VEL
LIN {X 0,Y 101.096,Z 465.382,A -85,B 0,C 180,E1 -29158.007,E2 -29158.007} C_VEL
LIN {X 0,Y 102.209,Z 468.432,A -85,B 0,C 180,E1 -29165.424,E2 -29165.424} C_VEL
LIN {X 0,Y 103.867,Z 472.471,A -85,B 0,C 180,E1 -29170.722,E2 -29170.722} C_VEL
LIN {X 0,Y 105.923,Z 477.148,A -85,B 0,C 180,E1 -29175.267,E2 -29175.267} C_VEL
LIN {X 0,Y 107.305,Z 481.04,A -85,B 0,C 180,E1 -29177.878,E2 -29177.878} C_VEL
LIN {X 0,Y 107.919,Z 484.03,A -85,B 0,C 180,E1 -29179.137,E2 -29179.137} C_VEL
LIN {X 0,Y 105.122,Z 509.213,A -85,B 0,C 180,E1 -29180.179,E2 -29180.179} C_VEL
LIN {X 0,Y 102.286,Z 522.485,A -85,B 0,C 180,E1 -29180.982,E2 -29180.982} C_VEL
LIN {X 0,Y 98.283,Z 535.432,A -85,B 0,C 180,E1 -29182.315,E2 -29182.315} C_VEL
LIN {X 0,Y 93.274,Z 547.246,A -85,B 0,C 180,E1 -29183.996,E2 -29183.996} C_VEL
LIN {X 0,Y 87.281,Z 558.646,A -85,B 0,C 180,E1 -29186.391,E2 -29186.391} C_VEL
LIN {X 0,Y 80.726,Z 568.896,A -85,B 0,C 180,E1 -29189.475,E2 -29189.475} C_VEL
LIN {X 0,Y 73.899,Z 578.136,A -85,B 0,C 180,E1 -29193.682,E2 -29193.682} C_VEL
LIN {X 0,Y 66.788,Z 586.453,A -85,B 0,C 180,E1 -29199.15,E2 -29199.15} C_VEL
LIN {X 0,Y 60.722,Z 593.23,A -85,B 0,C 180,E1 -29206.018,E2 -29206.018} C_VEL
LIN {X 0,Y 55.119,Z 599.219,A -85,B 0,C 180,E1 -29214.987,E2 -29214.987} C_VEL
LIN {X 0,Y 51.054,Z 603.933,A -85,B 0,C 180,E1 -29225.609,E2 -29225.609} C_VEL
LIN {X 0,Y 48.945,Z 607.519,A -85,B 0,C 180,E1 -29237.562,E2 -29237.562} C_VEL
LIN {X 0,Y 48.724,Z 610.064,A -85,B 0,C 180,E1 -29250,E2 -29250} C_VEL
LIN {X 0,Y 48.716,Z 611.189,A -85,B 0,C 180,E1 -29258.295,E2 -29258.295} C_VEL
LIN {X 0,Y 51.171,Z 612.162,A -85,B 0,C 180,E1 -29274.332,E2 -29274.332} C_VEL
LIN {X 0,Y 57.089,Z 611.624,A -85,B 0,C 180,E1 -29287.989,E2 -29287.989} C_VEL
LIN {X 0,Y 61.137,Z 610.758,A -85,B 0,C 180,E1 -29293.607,E2 -29293.607} C_VEL
LIN {X 0,Y 70.642,Z 607.818,A -85,B 0,C 180,E1 -29302.739,E2 -29302.739} C_VEL
LIN {X 0,Y 78.672,Z 604.502,A -85,B 0,C 180,E1 -29308.064,E2 -29308.064} C_VEL
LIN {X 0,Y 87.27,Z 600.145,A -85,B 0,C 180,E1 -29312.353,E2 -29312.353} C_VEL
LIN {X 0,Y 97.882,Z 593.607,A -85,B 0,C 180,E1 -29316.268,E2 -29316.268} C_VEL
LIN {X 0,Y 107.32,Z 586.46,A -85,B 0,C 180,E1 -29318.933,E2 -29318.933} C_VEL
LIN {X 0,Y 116.952,Z 577.596,A -85,B 0,C 180,E1 -29321.164,E2 -29321.164} C_VEL
LIN {X 0,Y 125.136,Z 568.523,A -85,B 0,C 180,E1 -29322.697,E2 -29322.697} C_VEL
LIN {X 0,Y 132.609,Z 558.518,A -85,B 0,C 180,E1 -29323.856,E2 -29323.856} C_VEL
LIN {X 0,Y 139.254,Z 547.427,A -85,B 0,C 180,E1 -29324.839,E2 -29324.839} C_VEL
LIN {X 0,Y 145.158,Z 534.987,A -85,B 0,C 180,E1 -29325.534,E2 -29325.534} C_VEL
LIN {X 0,Y 149.527,Z 522.505,A -85,B 0,C 180,E1 -29326.086,E2 -29326.086} C_VEL
LIN {X 0,Y 149.988,Z 520.775,A -85,B 0,C 180,E1 -29326.184,E2 -29326.184} C_VEL
LIN {X 0,Y 149.916,Z 517.927,A -85,B 0,C 180,E1 -29328.337,E2 -29328.337} C_VEL
LIN {X 0,Y 149.636,Z 516.575,A -85,B 0,C 180,E1 -29330.313,E2 -29330.313} C_VEL
LIN {X 0,Y 149.381,Z 514.562,A -85,B 0,C 180,E1 -29334.601,E2 -29334.601} C_VEL
LIN {X 0,Y 149.366,Z 514.597,A -85,B 0,C 180,E1 -29337.641,E2 -29337.641} C_VEL
LIN {X 0,Y 149.575,Z 516.823,A -85,B 0,C 180,E1 -29342.189,E2 -29342.189} C_VEL
LIN {X 0,Y 149.913,Z 519.718,A -85,B 0,C 180,E1 -29345.549,E2 -29345.549} C_VEL
LIN {X 0,Y 145.67,Z 532.222,A -85,B 0,C 180,E1 -29346.326,E2 -29346.326} C_VEL
LIN {X 0,Y 139.903,Z 544.572,A -85,B 0,C 180,E1 -29347.201,E2 -29347.201} C_VEL
LIN {X 0,Y 134.839,Z 553.246,A -85,B 0,C 180,E1 -29347.994,E2 -29347.994} C_VEL
LIN {X 0,Y 133.683,Z 555.048,A -85,B 0,C 180,E1 -29348.196,E2 -29348.196} C_VEL
LIN {X 0,Y 130.297,Z 559.857,A -85,B 0,C 180,E1 -29348.51,E2 -29348.51} C_VEL
LIN {X 0,Y 123.865,Z 567.424,A -85,B 0,C 180,E1 -29348.4,E2 -29348.4} C_VEL
LIN {X 0,Y 116.867,Z 574.437,A -85,B 0,C 180,E1 -29348.387,E2 -29348.387} C_VEL
LIN {X 0,Y 112.603,Z 578.373,A -85,B 0,C 180,E1 -29348.933,E2 -29348.933} C_VEL
LIN {X 0,Y 102.161,Z 586.969,A -85,B 0,C 180,E1 -29351.396,E2 -29351.396} C_VEL
LIN {X 0,Y 94.073,Z 592.453,A -85,B 0,C 180,E1 -29353.789,E2 -29353.789} C_VEL
LIN {X 0,Y 84.593,Z 597.782,A -85,B 0,C 180,E1 -29357.177,E2 -29357.177} C_VEL
LIN {X 0,Y 75.468,Z 601.901,A -85,B 0,C 180,E1 -29361.372,E2 -29361.372} C_VEL
LIN {X 0,Y 69.628,Z 604.049,A -85,B 0,C 180,E1 -29364.714,E2 -29364.714} C_VEL
LIN {X 0,Y 64.066,Z 605.713,A -85,B 0,C 180,E1 -29368.648,E2 -29368.648} C_VEL
LIN {X 0,Y 54.127,Z 607.811,A -85,B 0,C 180,E1 -29378.827,E2 -29378.827} C_VEL
LIN {X 0,Y 49.943,Z 608.217,A -85,B 0,C 180,E1 -29385.285,E2 -29385.285} C_VEL
LIN {X 0,Y 46.433,Z 608.219,A -85,B 0,C 180,E1 -29392.741,E2 -29392.741} C_VEL
LIN {X 0,Y 42.001,Z 607.063,A -85,B 0,C 180,E1 -29410.449,E2 -29410.449} C_VEL
LIN {X 0,Y 41.397,Z 605.842,A -85,B 0,C 180,E1 -29420.226,E2 -29420.226} C_VEL
LIN {X 0,Y 42.194,Z 603.837,A -85,B 0,C 180,E1 -29431.942,E2 -29431.942} C_VEL
LIN {X 0,Y 45.433,Z 599.707,A -85,B 0,C 180,E1 -29448.021,E2 -29448.021} C_VEL
LIN {X 0,Y 50.289,Z 595.056,A -85,B 0,C 180,E1 -29459.283,E2 -29459.283} C_VEL
LIN {X 0,Y 57.739,Z 588.056,A -85,B 0,C 180,E1 -29469.718,E2 -29469.718} C_VEL
LIN {X 0,Y 65.198,Z 580.487,A -85,B 0,C 180,E1 -29476.685,E2 -29476.685} C_VEL
LIN {X 0,Y 71.983,Z 572.738,A -85,B 0,C 180,E1 -29481.357,E2 -29481.357} C_VEL
LIN {X 0,Y 79.939,Z 562.19,A -85,B 0,C 180,E1 -29485.508,E2 -29485.508} C_VEL
LIN {X 0,Y 86.665,Z 551.457,A -85,B 0,C 180,E1 -29488.372,E2 -29488.372} C_VEL
LIN {X 0,Y 91.92,Z 541.058,A -85,B 0,C 180,E1 -29490.422,E2 -29490.422} C_VEL
LIN {X 0,Y 96.738,Z 528.997,A -85,B 0,C 180,E1 -29492.081,E2 -29492.081} C_VEL
LIN {X 0,Y 100.603,Z 515.742,A -85,B 0,C 180,E1 -29493.383,E2 -29493.383} C_VEL
LIN {X 0,Y 102.936,Z 503.639,A -85,B 0,C 180,E1 -29494.154,E2 -29494.154} C_VEL
LIN {X 0,Y 104.911,Z 485.931,A -85,B 0,C 180,E1 -29494.875,E2 -29494.875} C_VEL
LIN {X 0,Y 103.111,Z 480.753,A -85,B 0,C 180,E1 -29499.031,E2 -29499.031} C_VEL
LIN {X 0,Y 101.768,Z 477.532,A -85,B 0,C 180,E1 -29502.931,E2 -29502.931} C_VEL
LIN {X 0,Y 100.885,Z 475.132,A -85,B 0,C 180,E1 -29506.606,E2 -29506.606} C_VEL
LIN {X 0,Y 100.167,Z 471.966,A -85,B 0,C 180,E1 -29514.775,E2 -29514.775} C_VEL
LIN {X 0,Y 100.195,Z 471.847,A -85,B 0,C 180,E1 -29516.229,E2 -29516.229} C_VEL
LIN {X 0,Y 101.059,Z 475.341,A -85,B 0,C 180,E1 -29524.486,E2 -29524.486} C_VEL
LIN {X 0,Y 102.436,Z 479.112,A -85,B 0,C 180,E1 -29529.502,E2 -29529.502} C_VEL
LIN {X 0,Y 104.201,Z 483.751,A -85,B 0,C 180,E1 -29533.933,E2 -29533.933} C_VEL
LIN {X 0,Y 104.915,Z 486.226,A -85,B 0,C 180,E1 -29535.541,E2 -29535.541} C_VEL
LIN {X 0,Y 104.988,Z 486.629,A -85,B 0,C 180,E1 -29535.726,E2 -29535.726} C_VEL
LIN {X 0,Y 102.227,Z 509.668,A -85,B 0,C 180,E1 -29536.59,E2 -29536.59} C_VEL
LIN {X 0,Y 99.225,Z 523.04,A -85,B 0,C 180,E1 -29537.358,E2 -29537.358} C_VEL
LIN {X 0,Y 95.003,Z 535.86,A -85,B 0,C 180,E1 -29538.593,E2 -29538.593} C_VEL
LIN {X 0,Y 89.82,Z 547.52,A -85,B 0,C 180,E1 -29540.128,E2 -29540.128} C_VEL
LIN {X 0,Y 83.573,Z 558.806,A -85,B 0,C 180,E1 -29542.33,E2 -29542.33} C_VEL
LIN {X 0,Y 76.714,Z 568.939,A -85,B 0,C 180,E1 -29545.223,E2 -29545.223} C_VEL
LIN {X 0,Y 68.776,Z 578.941,A -85,B 0,C 180,E1 -29549.708,E2 -29549.708} C_VEL
LIN {X 0,Y 61.75,Z 586.486,A -85,B 0,C 180,E1 -29554.683,E2 -29554.683} C_VEL
LIN {X 0,Y 54.631,Z 593.675,A -85,B 0,C 180,E1 -29562.295,E2 -29562.295} C_VEL
LIN {X 0,Y 49.439,Z 598.602,A -85,B 0,C 180,E1 -29570.232,E2 -29570.232} C_VEL
LIN {X 0,Y 44.647,Z 603.377,A -85,B 0,C 180,E1 -29581.821,E2 -29581.821} C_VEL
LIN {X 0,Y 42.013,Z 607.02,A -85,B 0,C 180,E1 -29595.468,E2 -29595.468} C_VEL
LIN {X 0,Y 41.617,Z 609.618,A -85,B 0,C 180,E1 -29610,E2 -29610} C_VEL
LIN {X 0,Y 41.68,Z 610.774,A -85,B 0,C 180,E1 -29619.707,E2 -29619.707} C_VEL
LIN {X 0,Y 42.719,Z 611.497,A -85,B 0,C 180,E1 -29629.21,E2 -29629.21} C_VEL
LIN {X 0,Y 47.775,Z 611.755,A -85,B 0,C 180,E1 -29646.044,E2 -29646.044} C_VEL
LIN {X 0,Y 56.184,Z 610.508,A -85,B 0,C 180,E1 -29658.635,E2 -29658.635} C_VEL
LIN {X 0,Y 66.559,Z 607.621,A -85,B 0,C 180,E1 -29667.64,E2 -29667.64} C_VEL
LIN {X 0,Y 75.148,Z 604.36,A -85,B 0,C 180,E1 -29672.677,E2 -29672.677} C_VEL
LIN {X 0,Y 84.208,Z 600.06,A -85,B 0,C 180,E1 -29676.641,E2 -29676.641} C_VEL
LIN {X 0,Y 95.243,Z 593.591,A -85,B 0,C 180,E1 -29680.187,E2 -29680.187} C_VEL
LIN {X 0,Y 104.974,Z 586.545,A -85,B 0,C 180,E1 -29682.556,E2 -29682.556} C_VEL
LIN {X 0,Y 114.863,Z 577.765,A -85,B 0,C 180,E1 -29684.505,E2 -29684.505} C_VEL
LIN {X 0,Y 124.061,Z 567.817,A -85,B 0,C 180,E1 -29685.953,E2 -29685.953} C_VEL
LIN {X 0,Y 131.661,Z 557.697,A -85,B 0,C 180,E1 -29686.946,E2 -29686.946} C_VEL
LIN {X 0,Y 138.384,Z 546.57,A -85,B 0,C 180,E1 -29687.771,E2 -29687.771} C_VEL
LIN {X 0,Y 143.558,Z 535.882,A -85,B 0,C 180,E1 -29688.263,E2 -29688.263} C_VEL
LIN {X 0,Y 147.342,Z 525.849,A -85,B 0,C 180,E1 -29688.676,E2 -29688.676} C_VEL
LIN {X 0,Y 147.684,Z 524.489,A -85,B 0,C 180,E1 -29689.027,E2 -29689.027} C_VEL
LIN {X 0,Y 147.493,Z 522.812,A -85,B 0,C 180,E1 -29691.782,E2 -29691.782} C_VEL
LIN {X 0,Y 147.482,Z 521.366,A -85,B 0,C 180,E1 -29695.217,E2 -29695.217} C_VEL
LIN {X 0,Y 147.476,Z 521.37,A -85,B 0,C 180,E1 -29697.269,E2 -29697.269} C_VEL
LIN {X 0,Y 147.37,Z 522.586,A -85,B 0,C 180,E1 -29700.001,E2 -29700.001} C_VEL
LIN {X 0,Y 147.397,Z 524.623,A -85,B 0,C 180,E1 -29703.075,E2 -29703.075} C_VEL
LIN {X 0,Y 143.362,Z 535.225,A -85,B 0,C 180,E1 -29703.729,E2 -29703.729} C_VEL
LIN {X 0,Y 137.458,Z 547.058,A -85,B 0,C 180,E1 -29704.457,E2 -29704.457} C_VEL
LIN {X 0,Y 130.603,Z 557.83,A -85,B 0,C 180,E1 -29705.44,E2 -29705.44} C_VEL
LIN {X 0,Y 122.524,Z 568.181,A -85,B 0,C 180,E1 -29706.941,E2 -29706.941} C_VEL
LIN {X 0,Y 113.751,Z 577.336,A -85,B 0,C 180,E1 -29708.691,E2 -29708.691} C_VEL
LIN {X 0,Y 112.603,Z 578.373,A -85,B 0,C 180,E1 -29708.933,E2 -29708.933} C_VEL
LIN {X 0,Y 108.163,Z 582.163,A -85,B 0,C 180,E1 -29709.546,E2 -29709.546} C_VEL
LIN {X 0,Y 100.1,Z 587.978,A -85,B 0,C 180,E1 -29709.771,E2 -29709.771} C_VEL
LIN {X 0,Y 91.677,Z 593.104,A -85,B 0,C 180,E1 -29710.129,E2 -29710.129} C_VEL
LIN {X 0,Y 86.714,Z 595.837,A -85,B 0,C 180,E1 -29711.099,E2 -29711.099} C_VEL
LIN {X 0,Y 76.309,Z 600.794,A -85,B 0,C 180,E1 -29714.756,E2 -29714.756} C_VEL
LIN {X 0,Y 66.925,Z 604.236,A -85,B 0,C 180,E1 -29719.073,E2 -29719.073} C_VEL
LIN {X 0,Y 60.927,Z 605.934,A -85,B 0,C 180,E1 -29722.664,E2 -29722.664} C_VEL
LIN {X 0,Y 49.899,Z 608.088,A -85,B 0,C 180,E1 -29732.323,E2 -29732.323} C_VEL
LIN {X 0,Y 45.082,Z 608.544,A -85,B 0,C 180,E1 -29738.79,E2 -29738.79} C_VEL
LIN {X 0,Y 40.904,Z 608.573,A -85,B 0,C 180,E1 -29746.587,E2 -29746.587} C_VEL
LIN {X 0,Y 35.294,Z 607.47,A -85,B 0,C 180,E1 -29766.531,E2 -29766.531} C_VEL
LIN {X 0,Y 34.334,Z 606.298,A -85,B 0,C 180,E1 -29778.189,E2 -29778.189} C_VEL
LIN {X 0,Y 35.22,Z 604.081,A -85,B 0,C 180,E1 -29793.811,E2 -29793.811} C_VEL
LIN {X 0,Y 38.761,Z 600.264,A -85,B 0,C 180,E1 -29811.261,E2 -29811.261} C_VEL
LIN {X 0,Y 44.225,Z 595.68,A -85,B 0,C 180,E1 -29823.793,E2 -29823.793} C_VEL
LIN {X 0,Y 52.486,Z 588.746,A -85,B 0,C 180,E1 -29834.666,E2 -29834.666} C_VEL
LIN {X 0,Y 60.569,Z 581.255,A -85,B 0,C 180,E1 -29841.555,E2 -29841.555} C_VEL
LIN {X 0,Y 67.792,Z 573.605,A -85,B 0,C 180,E1 -29846.032,E2 -29846.032} C_VEL
LIN {X 0,Y 75.399,Z 564.27,A -85,B 0,C 180,E1 -29849.562,E2 -29849.562} C_VEL
LIN {X 0,Y 82.392,Z 553.903,A -85,B 0,C 180,E1 -29852.246,E2 -29852.246} C_VEL
LIN {X 0,Y 88.643,Z 542.426,A -85,B 0,C 180,E1 -29854.401,E2 -29854.401} C_VEL
LIN {X 0,Y 93.676,Z 530.687,A -85,B 0,C 180,E1 -29855.9,E2 -29855.9} C_VEL
LIN {X 0,Y 97.817,Z 517.402,A -85,B 0,C 180,E1 -29857.115,E2 -29857.115} C_VEL
LIN {X 0,Y 100.576,Z 504.035,A -85,B 0,C 180,E1 -29857.908,E2 -29857.908} C_VEL
LIN {X 0,Y 102.28,Z 489.565,A -85,B 0,C 180,E1 -29858.457,E2 -29858.457} C_VEL
LIN {X 0,Y 101.003,Z 485.618,A -85,B 0,C 180,E1 -29862.275,E2 -29862.275} C_VEL
LIN {X 0,Y 99.85,Z 482.051,A -85,B 0,C 180,E1 -29867.292,E2 -29867.292} C_VEL
LIN {X 0,Y 99.296,Z 479.008,A -85,B 0,C 180,E1 -29875.316,E2 -29875.316} C_VEL
LIN {X 0,Y 99.286,Z 479.568,A -85,B 0,C 180,E1 -29877.21,E2 -29877.21} C_VEL
LIN {X 0,Y 99.903,Z 482.025,A -85,B 0,C 180,E1 -29883.276,E2 -29883.276} C_VEL
LIN {X 0,Y 101.017,Z 485.635,A -85,B 0,C 180,E1 -29888.123,E2 -29888.123} C_VEL
LIN {X 0,Y 102.367,Z 489.777,A -85,B 0,C 180,E1 -29892.112,E2 -29892.112} C_VEL
LIN {X 0,Y 99.843,Z 509.674,A -85,B 0,C 180,E1 -29892.802,E2 -29892.802} C_VEL
LIN {X 0,Y 96.652,Z 523.305,A -85,B 0,C 180,E1 -29893.49,E2 -29893.49} C_VEL
LIN {X 0,Y 92.151,Z 536.288,A -85,B 0,C 180,E1 -29894.623,E2 -29894.623} C_VEL
LIN {X 0,Y 86.804,Z 547.792,A -85,B 0,C 180,E1 -29895.965,E2 -29895.965} C_VEL
LIN {X 0,Y 80.326,Z 558.956,A -85,B 0,C 180,E1 -29897.923,E2 -29897.923} C_VEL
LIN {X 0,Y 73.169,Z 568.98,A -85,B 0,C 180,E1 -29900.532,E2 -29900.532} C_VEL
LIN {X 0,Y 65.526,Z 578.096,A -85,B 0,C 180,E1 -29904.267,E2 -29904.267} C_VEL
LIN {X 0,Y 57.278,Z 586.409,A -85,B 0,C 180,E1 -29909.391,E2 -29909.391} C_VEL
LIN {X 0,Y 50.104,Z 592.992,A -85,B 0,C 180,E1 -29916.242,E2 -29916.242} C_VEL
LIN {X 0,Y 44.19,Z 597.985,A -85,B 0,C 180,E1 -29924.302,E2 -29924.302} C_VEL
LIN {X 0,Y 38.507,Z 602.82,A -85,B 0,C 180,E1 -29936.802,E2 -29936.802} C_VEL
LIN {X 0,Y 35.167,Z 606.521,A -85,B 0,C 180,E1 -29952.557,E2 -29952.557} C_VEL
LIN {X 0,Y 34.509,Z 609.172,A -85,B 0,C 180,E1 -29970,E2 -29970} C_VEL
LIN {X 0,Y 34.694,Z 610.353,A -85,B 0,C 180,E1 -29981.687,E2 -29981.687} C_VEL
LIN {X 0,Y 36.053,Z 611.122,A -85,B 0,C 180,E1 -29992.946,E2 -29992.946} C_VEL
LIN {X 0,Y 42.216,Z 611.432,A -85,B 0,C 180,E1 -30011.751,E2 -30011.751} C_VEL
LIN {X 0,Y 51.745,Z 610.248,A -85,B 0,C 180,E1 -30024.577,E2 -30024.577} C_VEL
LIN {X 0,Y 57.243,Z 609.04,A -85,B 0,C 180,E1 -30029.249,E2 -30029.249} C_VEL
LIN {X 0,Y 69.057,Z 605.402,A -85,B 0,C 180,E1 -30036.337,E2 -30036.337} C_VEL
LIN {X 0,Y 78.445,Z 601.512,A -85,B 0,C 180,E1 -30040.167,E2 -30040.167} C_VEL
LIN {X 0,Y 88.141,Z 596.521,A -85,B 0,C 180,E1 -30043.098,E2 -30043.098} C_VEL
LIN {X 0,Y 98.061,Z 590.279,A -85,B 0,C 180,E1 -30045.356,E2 -30045.356} C_VEL
LIN {X 0,Y 108.104,Z 582.517,A -85,B 0,C 180,E1 -30047.2,E2 -30047.2} C_VEL
LIN {X 0,Y 118.283,Z 572.824,A -85,B 0,C 180,E1 -30048.625,E2 -30048.625} C_VEL
LIN {X 0,Y 126.823,Z 562.829,A -85,B 0,C 180,E1 -30049.61,E2 -30049.61} C_VEL
LIN {X 0,Y 134.537,Z 551.541,A -85,B 0,C 180,E1 -30050.394,E2 -30050.394} C_VEL
LIN {X 0,Y 140.347,Z 540.934,A -85,B 0,C 180,E1 -30050.899,E2 -30050.899} C_VEL
LIN {X 0,Y 144.524,Z 531.399,A -85,B 0,C 180,E1 -30051.261,E2 -30051.261} C_VEL
LIN {X 0,Y 145.086,Z 529.733,A -85,B 0,C 180,E1 -30051.645,E2 -30051.645} C_VEL
LIN {X 0,Y 145.147,Z 528.431,A -85,B 0,C 180,E1 -30054.443,E2 -30054.443} C_VEL
LIN {X 0,Y 145.161,Z 528.153,A -85,B 0,C 180,E1 -30057.226,E2 -30057.226} C_VEL
LIN {X 0,Y 144.89,Z 529.679,A -85,B 0,C 180,E1 -30060.377,E2 -30060.377} C_VEL
LIN {X 0,Y 144.29,Z 531.365,A -85,B 0,C 180,E1 -30060.695,E2 -30060.695} C_VEL
LIN {X 0,Y 138.835,Z 543.187,A -85,B 0,C 180,E1 -30061.299,E2 -30061.299} C_VEL
LIN {X 0,Y 132.728,Z 553.544,A -85,B 0,C 180,E1 -30061.962,E2 -30061.962} C_VEL
LIN {X 0,Y 125.602,Z 563.395,A -85,B 0,C 180,E1 -30062.935,E2 -30062.935} C_VEL
LIN {X 0,Y 116.316,Z 573.857,A -85,B 0,C 180,E1 -30064.49,E2 -30064.49} C_VEL
LIN {X 0,Y 106.061,Z 583.027,A -85,B 0,C 180,E1 -30066.317,E2 -30066.317} C_VEL
LIN {X 0,Y 95.663,Z 590.568,A -85,B 0,C 180,E1 -30068.642,E2 -30068.642} C_VEL
LIN {X 0,Y 86.714,Z 595.837,A -85,B 0,C 180,E1 -30071.099,E2 -30071.099} C_VEL
LIN {X 0,Y 81.639,Z 598.406,A -85,B 0,C 180,E1 -30072.223,E2 -30072.223} C_VEL
LIN {X 0,Y 68.766,Z 603.399,A -85,B 0,C 180,E1 -30073.524,E2 -30073.524} C_VEL
LIN {X 0,Y 61.316,Z 605.505,A -85,B 0,C 180,E1 -30074.994,E2 -30074.994} C_VEL
LIN {X 0,Y 57.79,Z 606.307,A -85,B 0,C 180,E1 -30076.504,E2 -30076.504} C_VEL
LIN {X 0,Y 46.429,Z 608.363,A -85,B 0,C 180,E1 -30084.742,E2 -30084.742} C_VEL
LIN {X 0,Y 40.613,Z 608.879,A -85,B 0,C 180,E1 -30091.278,E2 -30091.278} C_VEL
LIN {X 0,Y 31.84,Z 608.594,A -85,B 0,C 180,E1 -30108.534,E2 -30108.534} C_VEL
LIN {X 0,Y 28.839,Z 607.873,A -85,B 0,C 180,E1 -30120.831,E2 -30120.831} C_VEL
LIN {X 0,Y 27.331,Z 606.751,A -85,B 0,C 180,E1 -30135.1,E2 -30135.1} C_VEL
LIN {X 0,Y 28.301,Z 604.326,A -85,B 0,C 180,E1 -30156.592,E2 -30156.592} C_VEL
LIN {X 0,Y 32.264,Z 600.807,A -85,B 0,C 180,E1 -30175.827,E2 -30175.827} C_VEL
LIN {X 0,Y 38.521,Z 596.29,A -85,B 0,C 180,E1 -30189.683,E2 -30189.683} C_VEL
LIN {X 0,Y 47.71,Z 589.436,A -85,B 0,C 180,E1 -30200.655,E2 -30200.655} C_VEL
LIN {X 0,Y 56.448,Z 582.019,A -85,B 0,C 180,E1 -30207.18,E2 -30207.18} C_VEL
LIN {X 0,Y 64.109,Z 574.458,A -85,B 0,C 180,E1 -30211.28,E2 -30211.28} C_VEL
LIN {X 0,Y 72.079,Z 565.275,A -85,B 0,C 180,E1 -30214.408,E2 -30214.408} C_VEL
LIN {X 0,Y 79.346,Z 555.063,A -85,B 0,C 180,E1 -30216.771,E2 -30216.771} C_VEL
LIN {X 0,Y 85.827,Z 543.771,A -85,B 0,C 180,E1 -30218.658,E2 -30218.658} C_VEL
LIN {X 0,Y 91.053,Z 532.302,A -85,B 0,C 180,E1 -30219.951,E2 -30219.951} C_VEL
LIN {X 0,Y 95.308,Z 519.64,A -85,B 0,C 180,E1 -30221.026,E2 -30221.026} C_VEL
LIN {X 0,Y 98.375,Z 506.077,A -85,B 0,C 180,E1 -30221.759,E2 -30221.759} C_VEL
LIN {X 0,Y 100.017,Z 493.45,A -85,B 0,C 180,E1 -30222.26,E2 -30222.26} C_VEL
LIN {X 0,Y 99.157,Z 490.505,A -85,B 0,C 180,E1 -30225.897,E2 -30225.897} C_VEL
LIN {X 0,Y 98.714,Z 488.726,A -85,B 0,C 180,E1 -30228.708,E2 -30228.708} C_VEL
LIN {X 0,Y 98.41,Z 486.25,A -85,B 0,C 180,E1 -30235.904,E2 -30235.904} C_VEL
LIN {X 0,Y 98.806,Z 488.855,A -85,B 0,C 180,E1 -30242.196,E2 -30242.196} C_VEL
LIN {X 0,Y 99.694,Z 492.322,A -85,B 0,C 180,E1 -30246.863,E2 -30246.863} C_VEL
LIN {X 0,Y 100.058,Z 493.675,A -85,B 0,C 180,E1 -30248.27,E2 -30248.27} C_VEL
LIN {X 0,Y 98.071,Z 508.855,A -85,B 0,C 180,E1 -30248.829,E2 -30248.829} C_VEL
LIN {X 0,Y 94.901,Z 522.32,A -85,B 0,C 180,E1 -30249.381,E2 -30249.381} C_VEL
LIN {X 0,Y 90.616,Z 534.717,A -85,B 0,C 180,E1 -30250.264,E2 -30250.264} C_VEL
LIN {X 0,Y 85.126,Z 546.478,A -85,B 0,C 180,E1 -30251.369,E2 -30251.369} C_VEL
LIN {X 0,Y 78.41,Z 557.817,A -85,B 0,C 180,E1 -30252.911,E2 -30252.911} C_VEL
LIN {X 0,Y 70.99,Z 568.041,A -85,B 0,C 180,E1 -30255.153,E2 -30255.153} C_VEL
LIN {X 0,Y 62.925,Z 577.252,A -85,B 0,C 180,E1 -30258.318,E2 -30258.318} C_VEL
LIN {X 0,Y 55.069,Z 584.842,A -85,B 0,C 180,E1 -30262.296,E2 -30262.296} C_VEL
LIN {X 0,Y 49.598,Z 589.559,A -85,B 0,C 180,E1 -30266.026,E2 -30266.026} C_VEL
LIN {X 0,Y 42.141,Z 595.47,A -85,B 0,C 180,E1 -30273.503,E2 -30273.503} C_VEL
LIN {X 0,Y 34.777,Z 600.779,A -85,B 0,C 180,E1 -30284.986,E2 -30284.986} C_VEL
LIN {X 0,Y 29.523,Z 604.905,A -85,B 0,C 180,E1 -30301.57,E2 -30301.57} C_VEL
LIN {X 0,Y 27.695,Z 607.047,A -85,B 0,C 180,E1 -30315.3,E2 -30315.3} C_VEL
LIN {X 0,Y 27.396,Z 608.725,A -85,B 0,C 180,E1 -30330,E2 -30330} C_VEL
LIN {X 0,Y 27.781,Z 609.932,A -85,B 0,C 180,E1 -30344.653,E2 -30344.653} C_VEL
LIN {X 0,Y 29.62,Z 610.736,A -85,B 0,C 180,E1 -30358.329,E2 -30358.329} C_VEL
LIN {X 0,Y 37.199,Z 611.109,A -85,B 0,C 180,E1 -30379.087,E2 -30379.087} C_VEL
LIN {X 0,Y 47.963,Z 609.976,A -85,B 0,C 180,E1 -30391.54,E2 -30391.54} C_VEL
LIN {X 0,Y 53.952,Z 608.818,A -85,B 0,C 180,E1 -30395.76,E2 -30395.76} C_VEL
LIN {X 0,Y 66.515,Z 605.232,A -85,B 0,C 180,E1 -30401.974,E2 -30401.974} C_VEL
LIN {X 0,Y 76.327,Z 601.398,A -85,B 0,C 180,E1 -30405.193,E2 -30405.193} C_VEL
LIN {X 0,Y 86.341,Z 596.467,A -85,B 0,C 180,E1 -30407.623,E2 -30407.623} C_VEL
LIN {X 0,Y 96.51,Z 590.291,A -85,B 0,C 180,E1 -30409.441,E2 -30409.441} C_VEL
LIN {X 0,Y 106.758,Z 582.636,A -85,B 0,C 180,E1 -30410.91,E2 -30410.91} C_VEL
LIN {X 0,Y 117.09,Z 573.042,A -85,B 0,C 180,E1 -30412.031,E2 -30412.031} C_VEL
LIN {X 0,Y 125.74,Z 563.163,A -85,B 0,C 180,E1 -30412.785,E2 -30412.785} C_VEL
LIN {X 0,Y 133.541,Z 552.088,A -85,B 0,C 180,E1 -30413.38,E2 -30413.38} C_VEL
LIN {X 0,Y 139.404,Z 541.693,A -85,B 0,C 180,E1 -30413.77,E2 -30413.77} C_VEL
LIN {X 0,Y 142.141,Z 535.899,A -85,B 0,C 180,E1 -30413.93,E2 -30413.93} C_VEL
LIN {X 0,Y 142.419,Z 535.164,A -85,B 0,C 180,E1 -30414.337,E2 -30414.337} C_VEL
LIN {X 0,Y 142.446,Z 534.826,A -85,B 0,C 180,E1 -30417.173,E2 -30417.173} C_VEL
LIN {X 0,Y 142.348,Z 535.101,A -85,B 0,C 180,E1 -30417.808,E2 -30417.808} C_VEL
LIN {X 0,Y 141.511,Z 537.037,A -85,B 0,C 180,E1 -30418.116,E2 -30418.116} C_VEL
LIN {X 0,Y 135.197,Z 548.98,A -85,B 0,C 180,E1 -30418.61,E2 -30418.61} C_VEL
LIN {X 0,Y 128.268,Z 559.35,A -85,B 0,C 180,E1 -30419.275,E2 -30419.275} C_VEL
LIN {X 0,Y 119.477,Z 570,A -85,B 0,C 180,E1 -30420.443,E2 -30420.443} C_VEL
LIN {X 0,Y 110.734,Z 578.552,A -85,B 0,C 180,E1 -30421.646,E2 -30421.646} C_VEL
LIN {X 0,Y 100.31,Z 586.844,A -85,B 0,C 180,E1 -30423.276,E2 -30423.276} C_VEL
LIN {X 0,Y 91.708,Z 592.474,A -85,B 0,C 180,E1 -30424.977,E2 -30424.977} C_VEL
LIN {X 0,Y 81.497,Z 597.935,A -85,B 0,C 180,E1 -30427.391,E2 -30427.391} C_VEL
LIN {X 0,Y 71.471,Z 602.175,A -85,B 0,C 180,E1 -30430.484,E2 -30430.484} C_VEL
LIN {X 0,Y 64.922,Z 604.408,A -85,B 0,C 180,E1 -30433.028,E2 -30433.028} C_VEL
LIN {X 0,Y 57.79,Z 606.307,A -85,B 0,C 180,E1 -30436.504,E2 -30436.504} C_VEL
LIN {X 0,Y 52.465,Z 607.433,A -85,B 0,C 180,E1 -30438.97,E2 -30438.97} C_VEL
LIN {X 0,Y 43.016,Z 608.73,A -85,B 0,C 180,E1 -30442.292,E2 -30442.292} C_VEL
LIN {X 0,Y 35.495,Z 609.203,A -85,B 0,C 180,E1 -30446.005,E2 -30446.005} C_VEL
LIN {X 0,Y 30.382,Z 609.214,A -85,B 0,C 180,E1 -30451.212,E2 -30451.212} C_VEL
LIN {X 0,Y 28.908,Z 609.101,A -85,B 0,C 180,E1 -30453.744,E2 -30453.744} C_VEL
LIN {X 0,Y 22.822,Z 608.276,A -85,B 0,C 180,E1 -30471.983,E2 -30471.983} C_VEL
LIN {X 0,Y 20.455,Z 607.193,A -85,B 0,C 180,E1 -30489.905,E2 -30489.905} C_VEL
LIN {X 0,Y 21.502,Z 604.552,A -85,B 0,C 180,E1 -30521.295,E2 -30521.295} C_VEL
LIN {X 0,Y 26.071,Z 601.339,A -85,B 0,C 180,E1 -30542.624,E2 -30542.624} C_VEL
LIN {X 0,Y 33.363,Z 596.884,A -85,B 0,C 180,E1 -30557.499,E2 -30557.499} C_VEL
LIN {X 0,Y 42.067,Z 591.221,A -85,B 0,C 180,E1 -30566.649,E2 -30566.649} C_VEL
LIN {X 0,Y 51.37,Z 584.133,A -85,B 0,C 180,E1 -30572.779,E2 -30572.779} C_VEL
LIN {X 0,Y 61.028,Z 575.31,A -85,B 0,C 180,E1 -30577.111,E2 -30577.111} C_VEL
LIN {X 0,Y 69.307,Z 566.244,A -85,B 0,C 180,E1 -30579.712,E2 -30579.712} C_VEL
LIN {X 0,Y 76.832,Z 556.222,A -85,B 0,C 180,E1 -30581.622,E2 -30581.622} C_VEL
LIN {X 0,Y 83.524,Z 545.109,A -85,B 0,C 180,E1 -30583.159,E2 -30583.159} C_VEL
LIN {X 0,Y 89.482,Z 532.502,A -85,B 0,C 180,E1 -30584.332,E2 -30584.332} C_VEL
LIN {X 0,Y 93.845,Z 519.798,A -85,B 0,C 180,E1 -30585.234,E2 -30585.234} C_VEL
LIN {X 0,Y 96.933,Z 506.496,A -85,B 0,C 180,E1 -30585.814,E2 -30585.814} C_VEL
LIN {X 0,Y 98.167,Z 497.783,A -85,B 0,C 180,E1 -30586.186,E2 -30586.186} C_VEL
LIN {X 0,Y 97.638,Z 495.418,A -85,B 0,C 180,E1 -30590.156,E2 -30590.156} C_VEL
LIN {X 0,Y 97.513,Z 493.509,A -85,B 0,C 180,E1 -30595.866,E2 -30595.866} C_VEL
LIN {X 0,Y 97.761,Z 495.718,A -85,B 0,C 180,E1 -30601.201,E2 -30601.201} C_VEL
LIN {X 0,Y 98.196,Z 497.958,A -85,B 0,C 180,E1 -30604.36,E2 -30604.36} C_VEL
LIN {X 0,Y 96.169,Z 511.287,A -85,B 0,C 180,E1 -30604.792,E2 -30604.792} C_VEL
LIN {X 0,Y 93.056,Z 523.338,A -85,B 0,C 180,E1 -30605.204,E2 -30605.204} C_VEL
LIN {X 0,Y 88.325,Z 536.145,A -85,B 0,C 180,E1 -30605.959,E2 -30605.959} C_VEL
LIN {X 0,Y 82.285,Z 548.336,A -85,B 0,C 180,E1 -30606.846,E2 -30606.846} C_VEL
LIN {X 0,Y 75.426,Z 559.2,A -85,B 0,C 180,E1 -30608.115,E2 -30608.115} C_VEL
LIN {X 0,Y 67.769,Z 569.067,A -85,B 0,C 180,E1 -30609.879,E2 -30609.879} C_VEL
LIN {X 0,Y 59.392,Z 578.056,A -85,B 0,C 180,E1 -30612.521,E2 -30612.521} C_VEL
LIN {X 0,Y 50.082,Z 586.323,A -85,B 0,C 180,E1 -30616.298,E2 -30616.298} C_VEL
LIN {X 0,Y 40.129,Z 593.79,A -85,B 0,C 180,E1 -30623.156,E2 -30623.156} C_VEL
LIN {X 0,Y 32.853,Z 598.557,A -85,B 0,C 180,E1 -30631.165,E2 -30631.165} C_VEL
LIN {X 0,Y 25.435,Z 603.118,A -85,B 0,C 180,E1 -30646.309,E2 -30646.309} C_VEL
LIN {X 0,Y 20.893,Z 606.574,A -85,B 0,C 180,E1 -30670.344,E2 -30670.344} C_VEL
LIN {X 0,Y 20.302,Z 608.279,A -85,B 0,C 180,E1 -30690,E2 -30690} C_VEL
LIN {X 0,Y 20.978,Z 609.51,A -85,B 0,C 180,E1 -30709.573,E2 -30709.573} C_VEL
LIN {X 0,Y 23.598,Z 610.341,A -85,B 0,C 180,E1 -30726.558,E2 -30726.558} C_VEL
LIN {X 0,Y 27.793,Z 610.771,A -85,B 0,C 180,E1 -30739.341,E2 -30739.341} C_VEL
LIN {X 0,Y 38.815,Z 610.433,A -85,B 0,C 180,E1 -30754.863,E2 -30754.863} C_VEL
LIN {X 0,Y 51.434,Z 608.589,A -85,B 0,C 180,E1 -30763.03,E2 -30763.03} C_VEL
LIN {X 0,Y 59.065,Z 606.731,A -85,B 0,C 180,E1 -30766.235,E2 -30766.235} C_VEL
LIN {X 0,Y 71.423,Z 602.673,A -85,B 0,C 180,E1 -30769.73,E2 -30769.73} C_VEL
LIN {X 0,Y 81.662,Z 598.179,A -85,B 0,C 180,E1 -30771.765,E2 -30771.765} C_VEL
LIN {X 0,Y 93.734,Z 591.423,A -85,B 0,C 180,E1 -30773.434,E2 -30773.434} C_VEL
LIN {X 0,Y 104.13,Z 584.089,A -85,B 0,C 180,E1 -30774.555,E2 -30774.555} C_VEL
LIN {X 0,Y 114.581,Z 575.015,A -85,B 0,C 180,E1 -30775.343,E2 -30775.343} C_VEL
LIN {X 0,Y 123.3,Z 565.629,A -85,B 0,C 180,E1 -30775.915,E2 -30775.915} C_VEL
LIN {X 0,Y 126.796,Z 561.287,A -85,B 0,C 180,E1 -30776.093,E2 -30776.093} C_VEL
LIN {X 0,Y 126.775,Z 561.304,A -85,B 0,C 180,E1 -30776.231,E2 -30776.231} C_VEL
LIN {X 0,Y 117.862,Z 571.578,A -85,B 0,C 180,E1 -30777.154,E2 -30777.154} C_VEL
LIN {X 0,Y 108.992,Z 579.905,A -85,B 0,C 180,E1 -30778.091,E2 -30778.091} C_VEL
LIN {X 0,Y 98.396,Z 588.021,A -85,B 0,C 180,E1 -30779.375,E2 -30779.375} C_VEL
LIN {X 0,Y 87.862,Z 594.498,A -85,B 0,C 180,E1 -30781.032,E2 -30781.032} C_VEL
LIN {X 0,Y 77.414,Z 599.594,A -85,B 0,C 180,E1 -30783.028,E2 -30783.028} C_VEL
LIN {X 0,Y 65.159,Z 604.114,A -85,B 0,C 180,E1 -30786.194,E2 -30786.194} C_VEL
LIN {X 0,Y 54.774,Z 606.81,A -85,B 0,C 180,E1 -30789.988,E2 -30789.988} C_VEL
LIN {X 0,Y 43.893,Z 608.638,A -85,B 0,C 180,E1 -30796.119,E2 -30796.119} C_VEL
LIN {X 0,Y 36.514,Z 609.224,A -85,B 0,C 180,E1 -30802.644,E2 -30802.644} C_VEL
LIN {X 0,Y 28.908,Z 609.101,A -85,B 0,C 180,E1 -30813.744,E2 -30813.744} C_VEL
LIN {X 0,Y 24.601,Z 608.787,A -85,B 0,C 180,E1 -30822.365,E2 -30822.365} C_VEL
LIN {X 0,Y 17.704,Z 607.626,A -85,B 0,C 180,E1 -30841.666,E2 -30841.666} C_VEL
LIN {X 0,Y 14.443,Z 606.212,A -85,B 0,C 180,E1 -30867.458,E2 -30867.458} C_VEL
LIN {X 0,Y 15.028,Z 604.781,A -85,B 0,C 180,E1 -30889.942,E2 -30889.942} C_VEL
LIN {X 0,Y 15.875,Z 604.207,A -85,B 0,C 180,E1 -30896.272,E2 -30896.272} C_VEL
LIN {X 0,Y 23.139,Z 600.527,A -85,B 0,C 180,E1 -30919.402,E2 -30919.402} C_VEL
LIN {X 0,Y 32.181,Z 595.741,A -85,B 0,C 180,E1 -30930.872,E2 -30930.872} C_VEL
LIN {X 0,Y 41.893,Z 589.702,A -85,B 0,C 180,E1 -30937.319,E2 -30937.319} C_VEL
LIN {X 0,Y 51.891,Z 582.198,A -85,B 0,C 180,E1 -30941.451,E2 -30941.451} C_VEL
LIN {X 0,Y 60.333,Z 574.542,A -85,B 0,C 180,E1 -30943.944,E2 -30943.944} C_VEL
LIN {X 0,Y 68.905,Z 565.184,A -85,B 0,C 180,E1 -30945.679,E2 -30945.679} C_VEL
LIN {X 0,Y 76.628,Z 554.801,A -85,B 0,C 180,E1 -30947.023,E2 -30947.023} C_VEL
LIN {X 0,Y 83.476,Z 543.303,A -85,B 0,C 180,E1 -30948.154,E2 -30948.154} C_VEL
LIN {X 0,Y 89.023,Z 531.259,A -85,B 0,C 180,E1 -30948.938,E2 -30948.938} C_VEL
LIN {X 0,Y 93.52,Z 517.775,A -85,B 0,C 180,E1 -30949.643,E2 -30949.643} C_VEL
LIN {X 0,Y 96.266,Z 505.439,A -85,B 0,C 180,E1 -30950.033,E2 -30950.033} C_VEL
LIN {X 0,Y 96.663,Z 502.684,A -85,B 0,C 180,E1 -30950.206,E2 -30950.206} C_VEL
LIN {X 0,Y 96.611,Z 500.713,A -85,B 0,C 180,E1 -30955.827,E2 -30955.827} C_VEL
LIN {X 0,Y 96.691,Z 502.447,A -85,B 0,C 180,E1 -30959.999,E2 -30959.999} C_VEL
LIN {X 0,Y 96.715,Z 502.682,A -85,B 0,C 180,E1 -30960.392,E2 -30960.392} C_VEL
LIN {X 0,Y 94.085,Z 516.116,A -85,B 0,C 180,E1 -30960.663,E2 -30960.663} C_VEL
LIN {X 0,Y 90.331,Z 528.349,A -85,B 0,C 180,E1 -30961.049,E2 -30961.049} C_VEL
LIN {X 0,Y 85.244,Z 540.322,A -85,B 0,C 180,E1 -30961.553,E2 -30961.553} C_VEL
LIN {X 0,Y 78.246,Z 552.904,A -85,B 0,C 180,E1 -30962.269,E2 -30962.269} C_VEL
LIN {X 0,Y 71.268,Z 562.845,A -85,B 0,C 180,E1 -30963.201,E2 -30963.201} C_VEL
LIN {X 0,Y 63.446,Z 571.991,A -85,B 0,C 180,E1 -30964.499,E2 -30964.499} C_VEL
LIN {X 0,Y 54.824,Z 580.388,A -85,B 0,C 180,E1 -30966.554,E2 -30966.554} C_VEL
LIN {X 0,Y 45.548,Z 587.821,A -85,B 0,C 180,E1 -30969.165,E2 -30969.165} C_VEL
LIN {X 0,Y 36.243,Z 594.162,A -85,B 0,C 180,E1 -30974.177,E2 -30974.177} C_VEL
LIN {X 0,Y 26.67,Z 599.606,A -85,B 0,C 180,E1 -30982.736,E2 -30982.736} C_VEL
LIN {X 0,Y 18.286,Z 603.849,A -85,B 0,C 180,E1 -30999.765,E2 -30999.765} C_VEL
LIN {X 0,Y 14.38,Z 606.091,A -85,B 0,C 180,E1 -31020.743,E2 -31020.743} C_VEL
LIN {X 0,Y 13.193,Z 607.832,A -85,B 0,C 180,E1 -31050,E2 -31050} C_VEL
LIN {X 0,Y 14.468,Z 609.088,A -85,B 0,C 180,E1 -31079.062,E2 -31079.062} C_VEL
LIN {X 0,Y 23.769,Z 610.414,A -85,B 0,C 180,E1 -31112.501,E2 -31112.501} C_VEL
LIN {X 0,Y 29.87,Z 610.464,A -85,B 0,C 180,E1 -31120.242,E2 -31120.242} C_VEL
LIN {X 0,Y 43.034,Z 609.43,A -85,B 0,C 180,E1 -31128.482,E2 -31128.482} C_VEL
LIN {X 0,Y 49.821,Z 608.346,A -85,B 0,C 180,E1 -31130.904,E2 -31130.904} C_VEL
